	garr_betriebsmeldungen[st_config_achse.i16_meld_startindex + 0] := FALSE;
	garr_betriebsmeldungen[st_config_achse.i16_meld_startindex + 1] := FALSE;
	garr_betriebsmeldungen[st_config_achse.i16_meld_startindex + 2] := FALSE;
	garr_betriebsmeldungen[st_config_achse.i16_meld_startindex + 3] := FALSE;
	garr_betriebsmeldungen[st_config_achse.i16_meld_startindex + 4] := FALSE;
	garr_betriebsmeldungen[st_config_achse.i16_meld_startindex + 5] := FALSE;
	garr_betriebsmeldungen[st_config_achse.i16_meld_startindex + 6] := FALSE;
	garr_betriebsmeldungen[st_config_achse.i16_meld_startindex + 7] := FALSE;
	garr_betriebsmeldungen[st_config_achse.i16_meld_startindex + 8] := FALSE;
	garr_betriebsmeldungen[st_config_achse.i16_meld_startindex + 9] := FALSE;
	garr_betriebsmeldungen[st_config_achse.i16_meld_startindex + 10] := FALSE;
	garr_betriebsmeldungen[st_config_achse.i16_meld_startindex + 11] := FALSE;
	garr_betriebsmeldungen[st_config_achse.i16_meld_startindex + 12] := FALSE;
	garr_betriebsmeldungen[st_config_achse.i16_meld_startindex + 13] := FALSE;
	garr_betriebsmeldungen[st_config_achse.i16_meld_startindex + 14] := FALSE;
	garr_betriebsmeldungen[st_config_achse.i16_meld_startindex + 15] := FALSE;
	garr_betriebsmeldungen[st_config_achse.i16_meld_startindex + 16] := FALSE;
	garr_betriebsmeldungen[st_config_achse.i16_meld_startindex + 17] := FALSE;
	garr_betriebsmeldungen[st_config_achse.i16_meld_startindex + 18] := FALSE;
	garr_betriebsmeldungen[st_config_achse.i16_meld_startindex + 19] := FALSE;
	garr_betriebsmeldungen[st_config_achse.i16_meld_startindex + 20] := FALSE;
	garr_betriebsmeldungen[st_config_achse.i16_meld_startindex + 21] := FALSE;
	garr_betriebsmeldungen[st_config_achse.i16_meld_startindex + 22] := FALSE;
	garr_betriebsmeldungen[st_config_achse.i16_meld_startindex + 23] := FALSE;
	garr_betriebsmeldungen[st_config_achse.i16_meld_startindex + 24] := FALSE;
	garr_betriebsmeldungen[st_config_achse.i16_meld_startindex + 25] := FALSE;
	garr_betriebsmeldungen[st_config_achse.i16_meld_startindex + 26] := FALSE;
	garr_betriebsmeldungen[st_config_achse.i16_meld_startindex + 27] := FALSE;
	garr_betriebsmeldungen[st_config_achse.i16_meld_startindex + 28] := FALSE;
	garr_betriebsmeldungen[st_config_achse.i16_meld_startindex + 29] := FALSE;
	garr_betriebsmeldungen[st_config_achse.i16_meld_startindex + 30] := FALSE;
	garr_betriebsmeldungen[st_config_achse.i16_meld_startindex + 31] := FALSE;
	garr_betriebsmeldungen[st_config_achse.i16_meld_startindex + 32] := FALSE;
	garr_betriebsmeldungen[st_config_achse.i16_meld_startindex + 33] := FALSE;
	garr_betriebsmeldungen[st_config_achse.i16_meld_startindex + 34] := FALSE;
	garr_betriebsmeldungen[st_config_achse.i16_meld_startindex + 35] := FALSE;
	garr_betriebsmeldungen[st_config_achse.i16_meld_startindex + 36] := FALSE;
	garr_betriebsmeldungen[st_config_achse.i16_meld_startindex + 37] := FALSE;
	garr_betriebsmeldungen[st_config_achse.i16_meld_startindex + 38] := FALSE;
	garr_betriebsmeldungen[st_config_achse.i16_meld_startindex + 39] := FALSE;
	garr_betriebsmeldungen[st_config_achse.i16_meld_startindex + 40] := FALSE;
	garr_betriebsmeldungen[st_config_achse.i16_meld_startindex + 41] := FALSE;
	garr_betriebsmeldungen[st_config_achse.i16_meld_startindex + 42] := FALSE;
	garr_betriebsmeldungen[st_config_achse.i16_meld_startindex + 43] := FALSE;
	garr_betriebsmeldungen[st_config_achse.i16_meld_startindex + 44] := FALSE;
	garr_betriebsmeldungen[st_config_achse.i16_meld_startindex + 45] := FALSE;
	garr_betriebsmeldungen[st_config_achse.i16_meld_startindex + 46] := FALSE;
	garr_betriebsmeldungen[st_config_achse.i16_meld_startindex + 47] := FALSE;
	garr_betriebsmeldungen[st_config_achse.i16_meld_startindex + 48] := FALSE;
	garr_betriebsmeldungen[st_config_achse.i16_meld_startindex + 49] := FALSE;
END_IF
END_PROGRAM

(* POU Maschine1720/WT Transport/ST_WT_Transport_Warteposition_1720, ST *)
PROGRAM ST_WT_Transport_Warteposition_1720
VAR_INPUT
	st_config								: struct_config;
	st_ctrl_in								: struct_ctrl_in;
	e_station_vorher_in_anforderung			: BOOL := FALSE;
	e_station_vorher_in_abgegeben			: BOOL := FALSE;
END_VAR
VAR_IN_OUT
	st_visu								: struct_visu;
END_VAR
VAR_OUTPUT
	st_ctrl_out							: struct_ctrl_out;
	a_station_vorher_out_erlaubnis			: BOOL := FALSE;
	a_station_vorher_out_angekommen		: BOOL := FALSE;
END_VAR
VAR
	fb_ton_uez							: TON;
	fb_ton_wz							: TON;
	fb_ton_quitt							: TON;
	fb_ton_wt_auf_wartepos				: TON;
	fb_tof_wt_auf_wartepos					: TOF;
	fb_r_trig_start							: R_TRIG;
	fb_r_trig_wartepos						: R_TRIG;
	fb_r_trig_wartepos_verlassen			: R_TRIG;
	fb_state_entry							: ST_StateEntry;
	sm_wt_hat_wartepos_nicht_verlassen	: BOOL := FALSE;
	sm_wt_hat_wartepos_ueberfahren		: BOOL := FALSE;
	bm_warte_anforderung					: BOOL := FALSE;
	bm_warte_wt_an_stopper				: BOOL := FALSE;
	bm_warte_beladepos_frei				: BOOL := FALSE;

	e_wt_auf_wartepos					AT %I* : BOOL;
	e_wt_wartepos_verlassen				AT %I* : BOOL;
END_VAR
(* Zeiten *)
fb_ton_uez(IN:= , PT:= , Q=>  , ET=> );
fb_ton_wz(IN:= , PT:= , Q=> , ET=> );
fb_ton_quitt(IN:= , PT:= t#100ms, Q=> , ET=> );

fb_ton_wt_auf_wartepos(IN:= e_wt_auf_wartepos, PT:= t#200ms, Q=> , ET=> );
fb_tof_wt_auf_wartepos(IN:= e_wt_auf_wartepos, PT:= t#200ms, Q=> , ET=> );

(* Flanken *)
fb_r_trig_wartepos(CLK:= e_wt_auf_wartepos, Q=> );
fb_r_trig_wartepos_verlassen(CLK:= e_wt_wartepos_verlassen, Q=> );
fb_r_trig_start(CLK:= st_ctrl_in.b_start, Q=> );

(* ==================================Toplevel=================================== *)
IF fb_state_entry.i16_next_step > INIT AND fb_state_entry.i16_next_step < FEHLER THEN
	(* Allgemeine Fehler *)
	IF st_ctrl_in.b_stop THEN
		fb_state_entry.i16_next_step := STOP;
	ELSIF zyl_wt_stopper_einlauf.st_ctrl.out.b_fehler THEN
		fb_state_entry.i16_next_step := FEHLER;
	(* Zylinder im Handbetrieb *)
	ELSIF gi16_betriebsart = HAND AND
		st_visu.st_zyl.i16_nr_zyl_im_handbetrieb = zyl_wt_stopper_einlauf.fb.st_config.i16_identnummer
		THEN
			fb_state_entry.i16_next_step := FEHLER;
	END_IF
END_IF

(* ============================Haupt-Schrittkette================================ *)
fb_state_entry(
	i16_next_step:= , 
	i16_pos:= 1,
	s_debugtext:= ,
	E=> ,
	X=> , 
	i16_step=> ,
	i16_last_step=> );

CASE fb_state_entry.i16_step OF
(*=======================================================*)
	INIT_OBJ:
		IF st_config.b_config_fertig THEN
			fb_state_entry.i16_next_step := INIT;
		END_IF

(*=======================================================*)
	INIT:
		IF fb_state_entry.E THEN
			fb_ton_wz.IN := FALSE;
			fb_ton_uez.IN := FALSE;
			fb_ton_quitt.IN := FALSE;
			st_ctrl_out.b_fehler := FALSE;
			st_ctrl_out.b_bereit := FALSE;
			st_ctrl_out.b_fertig := FALSE;
			st_ctrl_out.b_kontroller_start := FALSE;
			zyl_wt_stopper_einlauf.st_ctrl.in.b_einfahren := FALSE;
			zyl_wt_stopper_einlauf.st_ctrl.in.b_ausfahren := FALSE;
			sm_wt_hat_wartepos_nicht_verlassen := FALSE;
			sm_wt_hat_wartepos_ueberfahren := FALSE;
			bm_warte_anforderung := FALSE;
			bm_warte_wt_an_stopper := FALSE;
			bm_warte_beladepos_frei := FALSE;
			a_station_vorher_out_erlaubnis := FALSE;
			a_station_vorher_out_angekommen := FALSE;
		END_IF

		(*-----------------------Weiterschaltbedingungen----------------------------*)
		IF st_ctrl_in.b_init THEN
			zyl_wt_stopper_einlauf.st_ctrl.in.b_quittieren := FALSE;
			fb_state_entry.i16_next_step := 20;
		END_IF

(*=======================================================*)
	20: (* Initialisierung: Einlaufstopper ausfahren *)
		IF fb_state_entry.E THEN
			zyl_wt_stopper_einlauf.st_ctrl.in.b_ausfahren := TRUE;
		END_IF

		(*-----------------------Weiterschaltbedingungen----------------------------*)
		IF zyl_wt_stopper_einlauf.st_ctrl.out.b_ausgefahren THEN
			zyl_wt_stopper_einlauf.st_ctrl.in.b_ausfahren := FALSE;
			fb_state_entry.i16_next_step :=  BEREIT;
		END_IF

(*=======================================================*)
	BEREIT:	(* Warte auf Start von Kontroller *)
		IF fb_state_entry.E THEN
			st_ctrl_out.b_bereit := TRUE;
			st_ctrl_out.b_fertig := TRUE;
		END_IF

	(*-----------------------Weiterschaltbedingungen----------------------------*)
		IF st_config.b_station_aktiv OR st_config.b_station_in_simulation THEN
			(* WT Transport aktiv oder in Simulation *)
			IF st_ctrl_in.b_start THEN
			(* WT Transport gestartet *)
				st_ctrl_out.b_fertig := FALSE;
				fb_state_entry.i16_next_step := 110;
			END_IF
		ELSE
			fb_state_entry.i16_next_step := 500;
		END_IF

(*=======================================================*)
	110: (* Statische WT-Abfrage auf Warteposition nach der Initialisierung *)
		IF fb_state_entry.E THEN
			st_ctrl_out.b_kontroller_start := TRUE;
		END_IF

		IF NOT e_station_vorher_in_abgegeben THEN
			a_station_vorher_out_angekommen := FALSE;
		END_IF

		(*-----------------------Weiterschaltbedingungen----------------------------*)
		IF e_wt_auf_wartepos THEN
			st_ctrl_out.b_kontroller_start := FALSE;
			fb_state_entry.i16_next_step := 140;
		ELSE	(* Kein WT da, deshalb einen holen *)
			st_ctrl_out.b_kontroller_start := FALSE;
			fb_state_entry.i16_next_step := 120;
		END_IF

(*=======================================================*)
	120: (* Kein WT da -> warte auf Anforderung von vorheriger Station *)
		IF fb_state_entry.E THEN
			st_ctrl_out.b_kontroller_start := TRUE;
			bm_warte_anforderung := TRUE;
		END_IF

		IF NOT e_station_vorher_in_abgegeben THEN
			a_station_vorher_out_angekommen := FALSE;
		END_IF

		(*-----------------------Weiterschaltbedingungen----------------------------*)
		IF e_station_vorher_in_anforderung THEN
			a_station_vorher_out_angekommen := FALSE;
			a_station_vorher_out_erlaubnis := TRUE;
			st_ctrl_out.b_kontroller_start := FALSE;
			bm_warte_anforderung := FALSE;
			fb_state_entry.i16_next_step := 130;
		END_IF

(*=======================================================*)
	130: (* Warte bis WT an Stopper angekommen ist *)
		IF fb_state_entry.E THEN
			st_ctrl_out.b_kontroller_start := TRUE;
			bm_warte_wt_an_stopper := TRUE;
		END_IF

		(*-----------------------Weiterschaltbedingungen----------------------------*)
		IF fb_r_trig_wartepos.Q THEN
			a_station_vorher_out_erlaubnis := FALSE;
			a_station_vorher_out_angekommen := TRUE;
			st_ctrl_out.b_kontroller_start := FALSE;
			fb_ton_uez.IN := FALSE;
			bm_warte_wt_an_stopper := FALSE;
			fb_state_entry.i16_next_step := 140;
		END_IF

(*=======================================================*)
	140: (* WT ist da - Warten bis Beladeposition auf Bestücktisch frei ist *)
		IF fb_state_entry.E THEN
			zyl_wt_stopper_einlauf.st_ctrl.in.b_ausfahren := FALSE;
			zyl_wt_stopper_einlauf.st_ctrl.in.b_einfahren := FALSE;
			bm_warte_beladepos_frei := TRUE;
		END_IF

		(*-----------------------Weiterschaltbedingungen----------------------------*)
		IF NOT ST_WT_Transport_Beladen_1720.e_wt_auf_beladepos AND NOT axis_z_achse.st_ctrl.in.b_start THEN
			bm_warte_beladepos_frei := FALSE;
			fb_state_entry.i16_next_step := 150;
		ELSIF e_wt_wartepos_verlassen THEN
			(* Warteposition wurde unerlaubterweise überfahren *)
			sm_wt_hat_wartepos_ueberfahren := TRUE;
			fb_state_entry.i16_next_step := FEHLER;
		END_IF

(*=======================================================*)
	150: (* Bestücktisch ist frei -> Einlaufstopper einfahren *)
		IF fb_state_entry.E THEN
			zyl_wt_stopper_einlauf.st_ctrl.in.b_einfahren := TRUE;
		END_IF

		(*-----------------------Weiterschaltbedingungen----------------------------*)
		IF zyl_wt_stopper_einlauf.st_ctrl.out.b_eingefahren THEN
			zyl_wt_stopper_einlauf.st_ctrl.in.b_einfahren := FALSE;
			fb_state_entry.i16_next_step := 160;
		END_IF

(*=======================================================*)
	160: (* WT fährt weiter - Überwachung starten *)
		IF fb_state_entry.E THEN
			fb_ton_uez.PT := t#5s;
 			fb_ton_uez.IN := TRUE;
			st_ctrl_out.b_kontroller_start := TRUE;
		END_IF

		(*-----------------------Weiterschaltbedingungen----------------------------*)
		IF fb_r_trig_wartepos_verlassen.Q THEN
			fb_ton_uez.IN := FALSE;
			st_ctrl_out.b_kontroller_start := FALSE;
			fb_state_entry.i16_next_step := 170;
		ELSIF fb_ton_uez.Q THEN
			sm_wt_hat_wartepos_nicht_verlassen := TRUE;
			fb_state_entry.i16_next_step := FEHLER;
		END_IF

(*=======================================================*)
	170: (* Einlaufstopper ausfahren *)
		IF fb_state_entry.E THEN
			fb_ton_wz.IN := TRUE;
			fb_ton_wz.PT := t#1s;
			zyl_wt_stopper_einlauf.st_ctrl.in.b_ausfahren := TRUE;
		END_IF

		(*-----------------------Weiterschaltbedingungen----------------------------*)
		IF zyl_wt_stopper_einlauf.st_ctrl.out.b_ausgefahren AND fb_ton_wz.Q THEN
			zyl_wt_stopper_einlauf.st_ctrl.in.b_ausfahren := FALSE;
			fb_state_entry.i16_next_step := BEREIT;
			fb_ton_wz.IN := FALSE;
		END_IF

(*=======================================================*)
	500: (* Einlaufstopper einfahren, damit WTs auf Bestücktisch geschoben werden können. *)
		IF fb_state_entry.E THEN
			zyl_wt_stopper_einlauf.st_ctrl.in.b_einfahren := TRUE;
		END_IF

		(*-----------------------Weiterschaltbedingungen----------------------------*)
		IF zyl_wt_stopper_einlauf.st_ctrl.out.b_eingefahren THEN
			zyl_wt_stopper_einlauf.st_ctrl.in.b_einfahren := FALSE;
			fb_state_entry.i16_next_step :=  510;
		END_IF

(*=======================================================*)
	510:	(* Warte auf Konfigurationsänderung *)

	(*-----------------------Weiterschaltbedingungen----------------------------*)
		IF st_config.b_station_aktiv OR st_config.b_station_in_simulation THEN
			(* WT Transport aktiv oder in Simulation *)
			fb_state_entry.i16_next_step := BEREIT;
		END_IF

(*=======================================================*)
	FEHLER:
		IF fb_state_entry.E THEN
			st_ctrl_out.b_fehler := TRUE;
			fb_ton_quitt.IN := FALSE;
			zyl_wt_stopper_einlauf.st_ctrl.in.b_quittieren := FALSE;

			a_station_vorher_out_erlaubnis := FALSE;
			a_station_vorher_out_angekommen := FALSE;
		END_IF

		(*-----------------------Weiterschaltbedingungen----------------------------*)
		IF st_ctrl_in.b_quitt AND NOT fb_state_entry.E THEN
			st_ctrl_out.b_fehler := FALSE;
			zyl_wt_stopper_einlauf.st_ctrl.in.b_quittieren := TRUE;
			fb_ton_quitt.IN := TRUE;
		END_IF

		IF fb_ton_quitt.Q THEN
			fb_ton_quitt.IN := FALSE;
			fb_state_entry.i16_next_step := INIT;
		END_IF

(*=======================================================*)
	STOP:
		IF fb_state_entry.E THEN
			fb_ton_quitt.IN := FALSE;
			st_ctrl_out.b_kontroller_start := FALSE;
			zyl_wt_stopper_einlauf.st_ctrl.in.b_quittieren := FALSE;
			a_station_vorher_out_erlaubnis := FALSE;
			a_station_vorher_out_angekommen := FALSE;
		END_IF

		(*-----------------------Weiterschaltbedingungen----------------------------*)
		IF st_ctrl_in.b_quitt AND NOT fb_state_entry.E THEN
			fb_ton_quitt.IN := TRUE;
			zyl_wt_stopper_einlauf.st_ctrl.in.b_quittieren := TRUE;
		END_IF

		IF fb_ton_quitt.Q THEN
			fb_ton_quitt.IN := FALSE;
			fb_state_entry.i16_next_step := INIT;
		END_IF
END_CASE

fb_state_entry(
	i16_next_step:= ,
	i16_pos:= 2,
	s_debugtext:= ,
	E=> ,
	X=> ,
	i16_step=> ,
	i16_last_step=> );

IF st_config.b_config_fertig THEN
	(* Fehlermeldungen ab dem Startindex in das globale Störmeldungsarray schreiben *)
	garr_stoermeldungen[st_config.i16_meld_startindex + 0] := sm_wt_hat_wartepos_nicht_verlassen;
	garr_stoermeldungen[st_config.i16_meld_startindex + 1] := sm_wt_hat_wartepos_ueberfahren;
	garr_stoermeldungen[st_config.i16_meld_startindex + 2] := FALSE;
	garr_stoermeldungen[st_config.i16_meld_startindex + 3] := FALSE;
	garr_stoermeldungen[st_config.i16_meld_startindex + 4] := FALSE;
	garr_stoermeldungen[st_config.i16_meld_startindex + 5] := FALSE;
	garr_stoermeldungen[st_config.i16_meld_startindex + 6] := FALSE;
	garr_stoermeldungen[st_config.i16_meld_startindex + 7] := FALSE;
	garr_stoermeldungen[st_config.i16_meld_startindex + 8] := FALSE;
	garr_stoermeldungen[st_config.i16_meld_startindex + 9] := FALSE;
	garr_stoermeldungen[st_config.i16_meld_startindex + 10] := FALSE;
	garr_stoermeldungen[st_config.i16_meld_startindex + 11] := FALSE;
	garr_stoermeldungen[st_config.i16_meld_startindex + 12] := FALSE;
	garr_stoermeldungen[st_config.i16_meld_startindex + 13] := FALSE;
	garr_stoermeldungen[st_config.i16_meld_startindex + 14] := FALSE;
	garr_stoermeldungen[st_config.i16_meld_startindex + 15] := FALSE;
	garr_stoermeldungen[st_config.i16_meld_startindex + 16] := FALSE;
	garr_stoermeldungen[st_config.i16_meld_startindex + 17] := FALSE;
	garr_stoermeldungen[st_config.i16_meld_startindex + 18] := FALSE;
	garr_stoermeldungen[st_config.i16_meld_startindex + 19] := FALSE;
	
	garr_betriebsmeldungen[st_config.i16_meld_startindex + 0] := bm_warte_anforderung;
	garr_betriebsmeldungen[st_config.i16_meld_startindex + 1] := bm_warte_wt_an_stopper;
	garr_betriebsmeldungen[st_config.i16_meld_startindex + 2] := bm_warte_beladepos_frei;
	garr_betriebsmeldungen[st_config.i16_meld_startindex + 3] := FALSE;
	garr_betriebsmeldungen[st_config.i16_meld_startindex + 4] := FALSE;
	garr_betriebsmeldungen[st_config.i16_meld_startindex + 5] := FALSE;
	garr_betriebsmeldungen[st_config.i16_meld_startindex + 6] := FALSE;
	garr_betriebsmeldungen[st_config.i16_meld_startindex + 7] := FALSE;
	garr_betriebsmeldungen[st_config.i16_meld_startindex + 8] := FALSE;
	garr_betriebsmeldungen[st_config.i16_meld_startindex + 9] := FALSE;
	garr_betriebsmeldungen[st_config.i16_meld_startindex + 10] := FALSE;
	garr_betriebsmeldungen[st_config.i16_meld_startindex + 11] := FALSE;
	garr_betriebsmeldungen[st_config.i16_meld_startindex + 12] := FALSE;
	garr_betriebsmeldungen[st_config.i16_meld_startindex + 13] := FALSE;
	garr_betriebsmeldungen[st_config.i16_meld_startindex + 14] := FALSE;
	garr_betriebsmeldungen[st_config.i16_meld_startindex + 15] := FALSE;
	garr_betriebsmeldungen[st_config.i16_meld_startindex + 16] := FALSE;
	garr_betriebsmeldungen[st_config.i16_meld_startindex + 17] := FALSE;
	garr_betriebsmeldungen[st_config.i16_meld_startindex + 18] := FALSE;
	garr_betriebsmeldungen[st_config.i16_meld_startindex + 19] := FALSE;
END_IF
END_PROGRAM

(* POU Gemeinsamkeiten17xx/Werkzeug/ST_WkzAbsicherung, ST *)
PROGRAM ST_WkzAbsicherung
VAR_INPUT
	st_config								: struct_config;
	st_ctrl_in								: struct_ctrl_in;
END_VAR
VAR_IN_OUT
	st_visu								: struct_visu;
END_VAR
VAR_OUTPUT
	st_ctrl_out							: struct_ctrl_out;
END_VAR
VAR
	fb_ton_wz							: TON;
	fb_ton_uez							: TON;
	fb_ton_quitt							: TON;
	fb_state_entry							: ST_StateEntry;
	b_signalmerker_bestueckschieber_on		: BOOL := FALSE;
	b_signalmerker_bestueckschieber_off		: BOOL := FALSE;
	fb_r_trig_signal_bestueckschieber		: R_TRIG;
	fb_f_trig_signal_bestueckschieber		: F_TRIG;
	fb_r_trig_nocke_uw_bestueckschieber	: R_TRIG;
	fb_f_trig_nocke_uw_bestueckschieber	: F_TRIG;

	(* Eingänge *)
	(* BSV 1720 6-fach *)
	e_wkz_sicherung_niederhalter_li			AT %I* : BOOL;
	e_wkz_sicherung_faenger_li			AT %I* : BOOL;
	e_wkz_sicherung_abfallpodest_li		AT %I* : BOOL;
	e_wkz_sicherung_niederhalter_re		AT %I* : BOOL;
	e_wkz_sicherung_faenger_re			AT %I* : BOOL;
	e_wkz_sicherung_abfallpodest_re		AT %I* : BOOL;
	(* Erkennung/Kodierung für alte WKZ z.B. 1708alt *)
	e_kodierung_alt_wkz					AT %I* : BOOL;
	(* BSH 1700 *)
	e_wkz_sicherung_faenger				AT %I* : BOOL;
	e_bestueckschieber_ueberwachung		AT %I* : BOOL;

	(* Meldungen *)
	(* BSV 1720 6-fach *)
	sm_wkz_sicherung_niederhalter_li		: BOOL := FALSE;
	sm_wkz_sicherung_faenger_li			: BOOL := FALSE;
	sm_wkz_sicherung_abfallpodest_li		: BOOL := FALSE;
	sm_wkz_sicherung_niederhalter_re		: BOOL := FALSE;
	sm_wkz_sicherung_faenger_re			: BOOL := FALSE;
	sm_wkz_sicherung_abfallpodest_re		: BOOL := FALSE;
	(* BSH 1700 *)
	sm_wkz_sicherung_faenger				: BOOL := FALSE;
	sm_bestueckschieber_ueberwachung	: BOOL := FALSE;
	UW_Bestueckschieber_on: BOOL;
END_VAR
(* Zeiten *)
fb_ton_wz(IN:= , PT:= , Q=>  , ET=> );
fb_ton_uez(IN:= , PT:= , Q=>  , ET=> );
fb_ton_quitt(IN:= , PT:= t#100ms, Q=> , ET=> );

(* Flanken *)

fb_f_trig_nocke_uw_bestueckschieber(CLK:= nockenschaltwerk_bestueckachse.fb.arr_spur[SP_UW_BESTUECKSCHIEBER_ON], Q=> );
fb_r_trig_nocke_uw_bestueckschieber(CLK:= nockenschaltwerk_bestueckachse.fb.arr_spur[SP_UW_BESTUECKSCHIEBER_ON], Q=> );
fb_r_trig_signal_bestueckschieber(CLK:= e_bestueckschieber_ueberwachung, Q=> );
fb_f_trig_signal_bestueckschieber(CLK:= e_bestueckschieber_ueberwachung, Q=> );

UW_Bestueckschieber_on:=nockenschaltwerk_bestueckachse.fb.arr_spur[SP_UW_BESTUECKSCHIEBER_ON]; 	(*für Trace*)
(* Toplevel *)
IF fb_state_entry.i16_next_step > INIT AND fb_state_entry.i16_next_step < FEHLER THEN
	IF fb_state_entry.i16_next_step < STOP THEN
		IF st_ctrl_in.b_stop THEN
			fb_state_entry.i16_next_step := STOP;
		END_IF
	END_IF
END_IF

(* ======================================Schrittkette======================================== *)
fb_state_entry(
	i16_next_step:= ,
	i16_pos:= 1,
	s_debugtext:= ,
	E=> ,
	X=> ,
	i16_step=> ,
	i16_last_step=> );

CASE fb_state_entry.i16_step OF
(*=======================================================*)
	INIT_OBJ:
		IF st_config.b_config_fertig THEN
			fb_state_entry.i16_next_step := INIT;
		END_IF

(*=======================================================*)
	INIT:
		IF fb_state_entry.E THEN
			fb_ton_wz.IN := FALSE;
			fb_ton_uez.IN	:= FALSE;
			fb_ton_quitt.IN	 := FALSE;
			b_signalmerker_bestueckschieber_on := FALSE;
			b_signalmerker_bestueckschieber_off := FALSE;
			sm_wkz_sicherung_niederhalter_li := FALSE;
			sm_wkz_sicherung_faenger_li := FALSE;
			sm_wkz_sicherung_abfallpodest_li := FALSE;
			sm_wkz_sicherung_niederhalter_re := FALSE;
			sm_wkz_sicherung_faenger_re := FALSE;
			sm_wkz_sicherung_abfallpodest_re := FALSE;
			sm_wkz_sicherung_faenger := FALSE;
			sm_bestueckschieber_ueberwachung := FALSE;
			st_ctrl_out.b_fehler := FALSE;
			st_ctrl_out.b_bereit := FALSE;
			st_ctrl_out.b_fertig := FALSE;
			st_ctrl_out.b_einzelfertigung := FALSE;
		END_IF

		(*-----------------------Weiterschaltbedingungen----------------------------*)
		IF st_ctrl_in.b_init THEN
			fb_state_entry.i16_next_step := BEREIT;
		END_IF

(*=======================================================*)
	BEREIT:
		IF fb_state_entry.E THEN
			st_ctrl_out.b_bereit := TRUE;
		END_IF

		CASE gst_datensatz.st_md.i16_typ_zelle OF
			KEINE_ZELLE:
				;

			BESTUECKZELLE_1700:
				IF NOT gst_datensatz.st_md.b_wt_transport_simulation THEN
					IF NOT e_wkz_sicherung_faenger THEN
						sm_wkz_sicherung_faenger := TRUE;
						fb_state_entry.i16_next_step := FEHLER;
					END_IF

					IF ST_Virtuelle_Masterachse.fb_state_entry.i16_step >= BEREIT THEN
						IF gst_datensatz.st_bestueckprogramm.i16_b[ST_Virtuelle_Masterachse.i16_bestueckposzaehler] <> 0 THEN	(* Bei Umfahrung = 0 bewegt sich der Bestückschieber nicht *)
							(* Nocken werden in virtueller Bestückachse nach ein paar Hüben ausgeschaltet *)
							IF	(nockenschaltwerk_bestueckachse.fb.arr_spur[SP_UW_BESTUECKSCHIEBER_ON] AND  NOT e_bestueckschieber_ueberwachung) OR
								(nockenschaltwerk_bestueckachse.fb.arr_spur[SP_UW_BESTUECKSCHIEBER_OFF] AND e_bestueckschieber_ueberwachung)
								THEN
									sm_bestueckschieber_ueberwachung := TRUE;
									fb_state_entry.i16_next_step := FEHLER;
							END_IF
						END_IF
					END_IF


					(* Option: Flankenauswertung der GLS am Bestückschieber *)
(*					IF	nockenschaltwerk_bestueckachse.fb.arr_spur[SP_UW_BESTUECKSCHIEBER_ON] THEN
						IF 	fb_r_trig_signal_bestueckschieber.Q THEN
							b_signalmerker_bestueckschieber_on := TRUE;
						END_IF
						IF	 fb_f_trig_signal_bestueckschieber.Q THEN
							b_signalmerker_bestueckschieber_off := TRUE;
						END_IF
					END_IF

					(* Option: Beide setzen wenn Nocke abgeschaltet ist *)
					IF	NOT gst_datensatz.st_wkz.nockenschaltwerk_bestueckachse.arr_nocken[SP_UW_BESTUECKSCHIEBER_OFF].b_camvalid THEN
						b_signalmerker_bestueckschieber_on := TRUE;
						b_signalmerker_bestueckschieber_off := TRUE;
					END_IF

					IF 	fb_f_trig_nocke_uw_bestueckschieber.Q THEN

						IF 	b_signalmerker_bestueckschieber_off  AND
							b_signalmerker_bestueckschieber_on THEN
							b_signalmerker_bestueckschieber_on := FALSE;
							b_signalmerker_bestueckschieber_off := FALSE;
						ELSE
							sm_bestueckschieber_ueberwachung := TRUE;
							fb_state_entry.i16_next_step := FEHLER;
						END_IF
					END_IF
*)
				END_IF

			BESTUECKZELLE_1720:
				IF NOT gst_datensatz.st_md.b_wt_transport_simulation THEN
					IF e_kodierung_alt_wkz THEN
						(* BSV 1720 2-fach *)
						IF NOT  e_wkz_sicherung_faenger_li THEN
							sm_wkz_sicherung_faenger_li := TRUE;
							fb_state_entry.i16_next_step := FEHLER;
						END_IF
						IF NOT  e_wkz_sicherung_faenger_re THEN
							sm_wkz_sicherung_faenger_re := TRUE;
							fb_state_entry.i16_next_step := FEHLER;
						END_IF
					ELSE
						(* BSV 1720 6-fach *)
						IF	NOT ST_TippTasten.b_einfaedeln_aktiv THEN
							IF e_wkz_sicherung_niederhalter_li AND nockenschaltwerk_bestueckachse.fb.arr_spur[SP_UW_WKZ_NIEDERHALTER_LI] THEN
								sm_wkz_sicherung_niederhalter_li := TRUE;
								fb_state_entry.i16_next_step := 200;
							END_IF
							IF e_wkz_sicherung_niederhalter_re AND nockenschaltwerk_bestueckachse.fb.arr_spur[SP_UW_WKZ_NIEDERHALTER_RE] THEN
								sm_wkz_sicherung_niederhalter_re := TRUE;
								fb_state_entry.i16_next_step := 200;
							END_IF
						END_IF
						IF NOT  e_wkz_sicherung_faenger_li THEN
							sm_wkz_sicherung_faenger_li := TRUE;
							fb_state_entry.i16_next_step := FEHLER;
						END_IF
						IF NOT  e_wkz_sicherung_faenger_re THEN
							sm_wkz_sicherung_faenger_re := TRUE;
							fb_state_entry.i16_next_step := FEHLER;
						END_IF
						IF NOT e_wkz_sicherung_abfallpodest_li THEN
							sm_wkz_sicherung_abfallpodest_li := TRUE;
							fb_state_entry.i16_next_step := 200;
						END_IF
						IF NOT e_wkz_sicherung_abfallpodest_re THEN
							sm_wkz_sicherung_abfallpodest_re := TRUE;
							fb_state_entry.i16_next_step := 200;
						END_IF
					END_IF
				END_IF

			RASTERFOLIE:
				;
		END_CASE

(*=======================================================*)
	200:	(* Nur aktiv bei 1720 und WKZ-Absicherung 6-fach. Verzweigen nach Fehler erst, wenn OT erreicht wird - leichtere Fehlerbehebung. *)

		IF NOT gst_datensatz.st_md.b_wt_transport_simulation THEN
			(* BSV 1720 6-fach *)
			IF e_wkz_sicherung_niederhalter_li AND nockenschaltwerk_bestueckachse.fb.arr_spur[SP_UW_WKZ_NIEDERHALTER_LI] THEN
				sm_wkz_sicherung_niederhalter_li := TRUE;
			END_IF
			IF NOT  e_wkz_sicherung_faenger_li THEN
				sm_wkz_sicherung_faenger_li := TRUE;
				fb_state_entry.i16_next_step := FEHLER;
			END_IF
			IF NOT e_wkz_sicherung_abfallpodest_li THEN
				sm_wkz_sicherung_abfallpodest_li := TRUE;
			END_IF
			IF e_wkz_sicherung_niederhalter_re AND nockenschaltwerk_bestueckachse.fb.arr_spur[SP_UW_WKZ_NIEDERHALTER_RE] THEN
				sm_wkz_sicherung_niederhalter_re := TRUE;
			END_IF
			IF NOT  e_wkz_sicherung_faenger_re THEN
				sm_wkz_sicherung_faenger_re := TRUE;
				fb_state_entry.i16_next_step := FEHLER;
			END_IF
			IF NOT e_wkz_sicherung_abfallpodest_re THEN
				sm_wkz_sicherung_abfallpodest_re := TRUE;
			END_IF
		END_IF

		(*-----------------------Weiterschaltbedingungen----------------------------*)
		IF nockenschaltwerk_bestueckachse.fb.arr_spur[SP_OT]  THEN
			fb_state_entry.i16_next_step := FEHLER;
		END_IF

(*=======================================================*)
	FEHLER:
		IF fb_state_entry.E THEN
			st_ctrl_out.b_fehler := TRUE;
			fb_ton_quitt.IN := FALSE;
		END_IF

		(*-----------------------Weiterschaltbedingungen----------------------------*)
		IF st_ctrl_in.b_quitt AND NOT fb_state_entry.E THEN
			st_ctrl_out.b_fehler := FALSE;
			fb_ton_quitt.IN := TRUE;
		END_IF

		IF fb_ton_quitt.Q THEN
			fb_ton_quitt.IN := FALSE;
			fb_state_entry.i16_next_step := INIT;
		END_IF

(*=======================================================*)
	STOP:
		IF fb_state_entry.E THEN
			fb_ton_quitt.IN := FALSE;
		END_IF

		(*-----------------------Weiterschaltbedingungen----------------------------*)
		IF st_ctrl_in.b_quitt AND NOT fb_state_entry.E THEN
			fb_ton_quitt.IN := TRUE;
		END_IF

		IF fb_ton_quitt.Q THEN
			fb_ton_quitt.IN := FALSE;
			fb_state_entry.i16_next_step := INIT;
		END_IF
END_CASE

fb_state_entry(
	i16_next_step:= , 
	i16_pos:= 2,
	s_debugtext:= ,
	E=> , 
	X=> , 
	i16_step=> ,
	i16_last_step=> );

IF st_config.b_config_fertig THEN
	(* Fehlermeldungen und Betriebsmeldungen ab dem Startindex in die globalen Meldungsarrays schreiben *)
	garr_stoermeldungen[st_config.i16_meld_startindex + 0] := sm_wkz_sicherung_faenger;
	garr_stoermeldungen[st_config.i16_meld_startindex + 1] := sm_bestueckschieber_ueberwachung;
	garr_stoermeldungen[st_config.i16_meld_startindex + 2] := FALSE;
	garr_stoermeldungen[st_config.i16_meld_startindex + 3] := FALSE;
	garr_stoermeldungen[st_config.i16_meld_startindex + 4] := sm_wkz_sicherung_niederhalter_li;
	garr_stoermeldungen[st_config.i16_meld_startindex + 5] := sm_wkz_sicherung_faenger_li;
	garr_stoermeldungen[st_config.i16_meld_startindex + 6] := sm_wkz_sicherung_abfallpodest_li;
	garr_stoermeldungen[st_config.i16_meld_startindex + 7] := FALSE;
	garr_stoermeldungen[st_config.i16_meld_startindex + 8] := sm_wkz_sicherung_niederhalter_re;
	garr_stoermeldungen[st_config.i16_meld_startindex + 9] := sm_wkz_sicherung_faenger_re;
	garr_stoermeldungen[st_config.i16_meld_startindex + 10] := sm_wkz_sicherung_abfallpodest_re;
	garr_stoermeldungen[st_config.i16_meld_startindex + 11] := FALSE;
	garr_stoermeldungen[st_config.i16_meld_startindex + 12] := FALSE;
	garr_stoermeldungen[st_config.i16_meld_startindex + 13] := FALSE;
	garr_stoermeldungen[st_config.i16_meld_startindex + 14] := FALSE;
	garr_stoermeldungen[st_config.i16_meld_startindex + 15] := FALSE;
	garr_stoermeldungen[st_config.i16_meld_startindex + 16] := FALSE;
	garr_stoermeldungen[st_config.i16_meld_startindex + 17] := FALSE;
	garr_stoermeldungen[st_config.i16_meld_startindex + 18] := FALSE;
	garr_stoermeldungen[st_config.i16_meld_startindex + 19] := FALSE;
	
	garr_betriebsmeldungen[st_config.i16_meld_startindex + 0] := FALSE;
	garr_betriebsmeldungen[st_config.i16_meld_startindex + 1] := FALSE;
	garr_betriebsmeldungen[st_config.i16_meld_startindex + 2] := FALSE;
	garr_betriebsmeldungen[st_config.i16_meld_startindex + 3] := FALSE;
	garr_betriebsmeldungen[st_config.i16_meld_startindex + 4] := FALSE;
	garr_betriebsmeldungen[st_config.i16_meld_startindex + 5] := FALSE;
	garr_betriebsmeldungen[st_config.i16_meld_startindex + 6] := FALSE;
	garr_betriebsmeldungen[st_config.i16_meld_startindex + 7] := FALSE;
	garr_betriebsmeldungen[st_config.i16_meld_startindex + 8] := FALSE;
	garr_betriebsmeldungen[st_config.i16_meld_startindex + 9] := FALSE;
	garr_betriebsmeldungen[st_config.i16_meld_startindex + 10] := FALSE;
	garr_betriebsmeldungen[st_config.i16_meld_startindex + 11] := FALSE;
	garr_betriebsmeldungen[st_config.i16_meld_startindex + 12] := FALSE;
	garr_betriebsmeldungen[st_config.i16_meld_startindex + 13] := FALSE;
	garr_betriebsmeldungen[st_config.i16_meld_startindex + 14] := FALSE;
	garr_betriebsmeldungen[st_config.i16_meld_startindex + 15] := FALSE;
	garr_betriebsmeldungen[st_config.i16_meld_startindex + 16] := FALSE;
	garr_betriebsmeldungen[st_config.i16_meld_startindex + 17] := FALSE;
	garr_betriebsmeldungen[st_config.i16_meld_startindex + 18] := FALSE;
	garr_betriebsmeldungen[st_config.i16_meld_startindex + 19] := FALSE;
END_IF
END_PROGRAM

(* POU EPT Lib/Funktionen/DT_TO_SPECIALSTRING_YYYY_MM, ST *)
FUNCTION DT_TO_SPECIALSTRING_YYYY_MM : STRING
VAR_INPUT
	inDT					:	DT;
END_VAR
VAR

	TempString		:	STRING;
	SysTime				:	TIMESTRUCT;


	wYear					: WORD;
	wMonth				: WORD;
	wDay					: WORD;
	wHour					: WORD;
	wMin					: WORD;
	wSec					: WORD;
END_VAR
(*gVarStrSystemTime:=SYSTEMTIME_TO_STRING(gFB_GETLOCALSYSTEMTIME.systemTime);
gVarDTSystemtime:=SYSTEMTIME_TO_DT(gFB_GETLOCALSYSTEMTIME.SystemTime);
gVarSystemtime:=gFB_GETLOCALSYSTEMTIME.systemTime;
*)

SysTime:=DT_TO_SYSTEMTIME(inDT);

wYear:=SysTime.wYear;
wMonth:=SysTime.wMonth;
wDay:=SysTime.wDay;
wHour:=SysTime.wHour;
wMin:=SysTime.wMinute;
wSec:=SysTime.wSecond;
TempString:='';

TempString:=CONCAT(TempString ,WORD_TO_STRING(wYear));
TempString:=CONCAT(TempString ,'_');

IF wMonth<10 THEN	TempString:=CONCAT(TempString ,WORD_TO_STRING(0)); END_IF;
TempString:=CONCAT(TempString ,WORD_TO_STRING(wMonth));


DT_TO_SPECIALSTRING_YYYY_MM:=TempString;
END_FUNCTION

(* POU Gemeinsamkeiten17xx/Allgemeines/ST_Gesamthubzaehler, ST *)
PROGRAM ST_Gesamthubzaehler
VAR
	fb_tp_wz				: TP;
	fb_r_trig				: R_TRIG;
	a_Gesamthubzaehler	 AT %Q* : BOOL;
END_VAR
(* Erzeugung eines zeitkonstanten Zählersignals *)
fb_tp_wz(IN:= nockenschaltwerk_bestueckachse.fb.arr_spur[SP_OT], PT:= t#20ms, Q=> a_Gesamthubzaehler, ET=> );

(* Interner Bestückhubzähler der Maschine*)
fb_r_trig(CLK:= nockenschaltwerk_bestueckachse.fb.arr_spur[SP_OT], Q=> );

IF fb_r_trig.Q THEN
	gst_datensatz.st_md.i32_bestueckhubzaehler := gst_datensatz.st_md.i32_bestueckhubzaehler + 1;
	gst_datensatz.st_md.i32_werkzeughubzaehler := 	gst_datensatz.st_md.i32_werkzeughubzaehler +1;
END_IF

IF gst_datensatz.st_md.i32_bestueckhubzaehler > (EXPT(2,32)) OR gst_datensatz.st_md.i32_bestueckhubzaehler < 0 THEN
	gst_datensatz.st_md.i32_bestueckhubzaehler := 0;
END_IF
END_PROGRAM

(* POU Gemeinsamkeiten17xx/Allgemeines/ST_LampeMaterialMangel, ST *)
PROGRAM ST_LampeMaterialMangel
VAR_INPUT
	b_materialmangel		: ARRAY[0..7] OF BOOL;
END_VAR
VAR
	a_Lampe			AT %Q* : BOOL;
	fb_blinker			: ST_Blinker;
END_VAR
(* Blinken *)
(*schnell*)
IF 	b_materialmangel[1] 	THEN	(*Öl leer*)
fb_blinker(
	b_start:= TRUE,
	t_taktzeit_on:=t#500ms,
	t_taktzeit_off:=t#500ms,
	b_blinker_out=> );
END_IF
(*langsam*)
IF 	NOT b_materialmangel[1] AND	(*Öl leer*)
	( b_materialmangel[2] OR b_materialmangel[6] ) THEN	(*Stufe kleiner 10 or Korrektur X-Y zu hoch*)
fb_blinker(
	b_start:= TRUE,
	t_taktzeit_on:=t#1500ms,
	t_taktzeit_off:=t#1500ms,
	b_blinker_out=> );
END_IF


(* Materialmangel ist eingetreten *)
IF 	b_materialmangel[0] OR	(*Band leer*)
	b_materialmangel[1] OR	(*Öl leer*)
	b_materialmangel[2] OR	(*Stufe kleiner 10*)
	b_materialmangel[3] OR	(* Bandwechsel *)
	b_materialmangel[4] OR	(*Schaltschrank Temp*)
	b_materialmangel[5] OR	(* Band nicht abgescannt *)
	b_materialmangel[6] 		(* Korrektur X-Y Wert zu hoch *)
	THEN
		a_Lampe := fb_blinker.b_blinker_out OR b_materialmangel[0] OR b_materialmangel[3];

(* Es liegt kein Materialmangel vor *)
ELSE
	a_Lampe := FALSE;
END_IF
END_PROGRAM

(* POU EPT Lib/Funktionsbausteine/ST_Blinker, ST *)
FUNCTION_BLOCK ST_Blinker
VAR_INPUT
	b_start 		: BOOL;
	t_taktzeit_on	: TIME;
	t_taktzeit_off	: TIME;
END_VAR
VAR_OUTPUT
	b_blinker_out : BOOL;
END_VAR
VAR
	ton_on		: TON;
	ton_off		: TON;
END_VAR
ton_on(IN:=b_start AND NOT ton_off.Q , PT:=t_taktzeit_on , Q=>b_blinker_out , ET=> );
ton_off(IN:= ton_on.Q  , PT:=t_taktzeit_off , Q=> , ET=> );
END_FUNCTION_BLOCK

(* POU Gemeinsamkeiten17xx/Allgemeines/ST_Scope, ST *)
PROGRAM ST_Scope
VAR
	fb_ton_wz			: TON;
	fb_r_trig_bereit		: R_TRIG;
	fb_state_entry			: ST_StateEntry;

	fb_ScopeStop		: ScopeSetOffline;
	fb_ScopeOnline		: ScopeSetOnline;
	fb_ScopeExport		: ScopeViewExport;

	b_Stop				: BOOL;
	s_file_name			: STRING;
	pos					: INT;
	i					: INT;
	i32_error_id			:UDINT;
END_VAR

VAR CONSTANT
	s_path				: STRING:='C:\TwinCAT\Scope\';
END_VAR
(*===============================================================
   PRG: ST_Scope
  ---------------------------------------------------------------
   Auth: 		Werner Friedl
   Date: 		03.08.2016    						    
   Rev.: 		1.0
   Beschreibung:
	Mit diesem Programm wird das Scope automatisch gestartet und bei einem Fehler 
	ein Scopedatei mit aktueller Zeit im Verzeichnis "C:\TwinCAT\Scope\" abgespeichert. 

	-	zuerst muss ein Scope geöffnet und ein Projekt erstellt werden.
	-	Fehler für Stop eintragen	
	-	ST_ScopeStop startet das Scope bei "Anlage betriebsbereit"
	-	bei Fehler wird die Aufzeichnung nach 2sec gestoppt
	-	Auzeichnung	wird mit aktueller Zeit abgespeichert.	

hier Fehler für Stop einfügen============================================*)
(*b_Stop:=	ST_Bestueckachse.st_ctrl_out.b_fehler  OR
		axis_bestueckachse.st_ctrl.out.b_fehler ;*)

b_Stop:= (gi16_maschinenstatusinfo = STATUS_FEHLER);

(*=======================================================*)
fb_ton_wz(IN:=,PT:=T#2s);
fb_r_trig_bereit(CLK:= gi16_maschinenstatusinfo = STATUS_BETRIEBSBEREIT, Q=> );
fb_ScopeStop(bExecute:= , bBusy=> , bError=> , iErrorId=> );
fb_ScopeOnline(bExecute:= , bBusy=> , bError=> , iErrorId=> );
fb_ScopeExport(bExecute:=, sFilePath:=, tTimeout:=T#5s);

(*=======================================================*)
fb_state_entry(i16_pos:= 1, );

CASE fb_state_entry.i16_step OF
(*=======================================================*)
	INIT_OBJ:
		fb_state_entry.i16_next_step := INIT;

(*=======================================================*)
	INIT:
		IF	fb_state_entry.E THEN
			fb_ScopeOnline.bExecute:=FALSE;
			fb_ScopeStop.bExecute:=FALSE;
			fb_ScopeExport.bExecute:=FALSE;
		END_IF

		fb_state_entry.i16_next_step := BEREIT;


(*=======================================================*)
	BEREIT: (*warten auf betriebsbereit *)
		IF	fb_state_entry.E THEN
			b_Stop:=FALSE;
		END_IF

		IF	fb_r_trig_bereit.Q THEN
			fb_state_entry.i16_next_step := 110;
		END_IF


(*=======================================================*)
	110: (* Scope starten *)
		IF 	fb_state_entry.E THEN
			fb_ScopeOnline.bExecute:=TRUE;
		END_IF

		(*-----------------------Weiterschaltbedingungen----------------------------*)
		IF	fb_ScopeOnline.bBusy THEN
			fb_state_entry.i16_next_step := 120;
		END_IF

(*=======================================================*)
	120: (* Scope starten *)

		IF	NOT fb_ScopeOnline.bBusy THEN
			fb_state_entry.i16_next_step := 130;
			fb_ScopeOnline.bExecute:=FALSE;
		END_IF

		IF	fb_ScopeOnline.bError THEN
			i32_error_id:=fb_ScopeOnline.iErrorId;
			fb_state_entry.i16_next_step := FEHLER;
		END_IF

(*=======================================================*)
	130: (* warten auf Fehler *)
		IF	 fb_state_entry.E THEN
			fb_ton_wz.IN:=FALSE;
		END_IF

		fb_ton_wz.IN:=b_Stop ;
		fb_ScopeStop.bExecute:=fb_ton_wz.Q;


		IF	fb_ScopeStop.bBusy THEN
			fb_state_entry.i16_next_step := 140;
		END_IF

		IF	 fb_state_entry.X THEN
			fb_ton_wz.IN:=FALSE;
		END_IF
(*=======================================================*)
	140: (* Scope anhalten *)

		IF	NOT fb_ScopeStop.bBusy THEN
			fb_ScopeStop.bExecute:=FALSE;
			fb_state_entry.i16_next_step := 150;
		END_IF

		IF	fb_ScopeStop.bError THEN
			i32_error_id:=fb_ScopeStop.iErrorId;
			fb_state_entry.i16_next_step := FEHLER;
		END_IF

(*=======================================================*)
	150: (* Scope speichern *)
		IF 	fb_state_entry.E THEN
			s_file_name:=gstr_system_time;
			i:=0;
			FOR i := 1 TO 5  BY 1DO
				pos:=0;
				pos:=FIND(s_file_name,':');
				IF	pos > 0 THEN
					s_file_name:=REPLACE(s_file_name,'-',1,pos);
				END_IF
			END_FOR

			s_file_name:=CONCAT(s_file_name,'_Scope_View');
			s_file_name:=CONCAT(s_file_name,'.svw');

			fb_ScopeExport.sFilePath:=CONCAT(s_path,s_file_name);
			fb_ScopeExport.bExecute:=TRUE;
		END_IF

		(*-----------------------Weiterschaltbedingungen----------------------------*)
		IF	fb_ScopeExport.bBusy THEN
			fb_state_entry.i16_next_step := 160;
		END_IF


(*=======================================================*)
	160: (* Scope speichern *)

		IF	NOT fb_ScopeExport.bBusy THEN
			fb_state_entry.i16_next_step := BEREIT;
			fb_ScopeExport.bExecute:=FALSE;
		END_IF

		IF	fb_ScopeExport.bError THEN
			i32_error_id:=fb_ScopeExport.iErrorId;
			fb_state_entry.i16_next_step := FEHLER;
		END_IF

(*=======================================================*)
	FEHLER:	(*bei Fehler einfach weiter*)
		IF 	fb_state_entry.E THEN
			;
		END_IF
			fb_state_entry.i16_next_step := INIT;

END_CASE

fb_state_entry(i16_pos:= 2 );
END_PROGRAM

(* POU Gemeinsamkeiten17xx/Allgemeines/ST_Tuerverriegelung, ST *)
PROGRAM ST_Tuerverriegelung
VAR_INPUT
	e_quittiertaste						: BOOL;
END_VAR
VAR
	fb_ton_wz						: TON;
	fb_r_trig_quitt						: R_TRIG;
	fb_f_trig_quitt						: F_TRIG;
	fb_blinker						: ST_Blinker;
	a_tuerverriegelung_vorne			AT %Q* : BOOL;
	a_tuerverriegelung_hinten			AT %Q* : BOOL;
	e_kontakt_tuerverriegelung_vorne	AT %I* : BOOL;
	e_kontakt_tuerverriegelung_hinten	AT %I* : BOOL;
END_VAR
(* Blinken *)
fb_blinker(
	b_start:= TRUE,
	t_taktzeit_on:=t#500ms,
	t_taktzeit_off:=t#500ms,
	b_blinker_out=> );

(* Zeiten *)
fb_ton_wz(IN:= , PT:= t#3s, Q=> , ET=> );

(* Flanken *)
fb_r_trig_quitt(CLK:= e_quittiertaste, Q=> );
fb_f_trig_quitt(CLK:= e_quittiertaste, Q=> );

(* Ansteuerung der Türverriegelung vorne und hinten *)
CASE gi16_betriebsart OF
	HAND:
		a_tuerverriegelung_vorne := FALSE;
		a_tuerverriegelung_hinten := FALSE;
	TIPPEN, AUTO:
		IF 	gi16_maschinenstatusinfo = STATUS_BETRIEBSBEREIT OR
			gi16_maschinenstatusinfo = STATUS_FEHLER
			THEN
				(* Türen freigeben *)
				a_tuerverriegelung_vorne := FALSE;
				a_tuerverriegelung_hinten := FALSE;
		ELSE
			(* Türen verriegelt, wenn geschlossen *)
			IF NOT e_kontakt_tuerverriegelung_vorne THEN
				a_tuerverriegelung_vorne := TRUE;
			END_IF
			IF NOT e_kontakt_tuerverriegelung_hinten THEN
				a_tuerverriegelung_hinten := TRUE;
			END_IF
		END_IF
END_CASE
END_PROGRAM

(* POU Gemeinsamkeiten17xx/Bandeinzug/ST_Anwahl_Bandeinzug, ST *)
PROGRAM ST_Anwahl_Bandeinzug
VAR
	b_first_cycle 						: BOOL := TRUE;
	i16_typ_bandeinzug_visu			: enum_typ_bandeinzug_visu := KEIN_BANDEINZUG;
END_VAR
(*======================================================
   PRG: ExportResultString
 ------------------------------------------------------
   Auth: 		Werner Friedl    						 
   Date: 		07.03.2016    						     
   Rev.: 		1.0	
   Desc:		Damit bei unterschiedlichen Zellen (1700 oder 1720) nur die vorhandenen Bandwechsler in der Visu vorne angezeigt werden,
			müssen diese der Struktur "i16_typ_bandeinzug" zugewiesen werden.
   Historie:   1.0

 ========================================================*)
IF 	gi16_bbgen_auftrag = LESE_WKZ THEN
	b_first_cycle:=TRUE;
END_IF



IF	NOT b_first_cycle THEN

	CASE gst_datensatz.st_md.i16_typ_zelle OF
		KEINE_ZELLE:
			;

		BESTUECKZELLE_1700, RASTERFOLIE:
	
			CASE i16_typ_bandeinzug_visu OF

				KEIN_BANDEINZUG :
						gst_datensatz.st_wkz.i16_typ_bandeinzug:=KEIN_EINZUG;					;
				BANDEINZUG_1:
						gst_datensatz.st_wkz.i16_typ_bandeinzug:=BANDWECHSLER_V2;
				BANDEINZUG_2:
						gst_datensatz.st_wkz.i16_typ_bandeinzug:=SERVO;
				BANDEINZUG_3:
					;
			END_CASE

		BESTUECKZELLE_1720:

			CASE i16_typ_bandeinzug_visu OF
	
				KEIN_BANDEINZUG :
						gst_datensatz.st_wkz.i16_typ_bandeinzug:=KEIN_EINZUG;
				BANDEINZUG_1:
						gst_datensatz.st_wkz.i16_typ_bandeinzug:=STANDARD_2FACH_V2;
				BANDEINZUG_2:
					;
				BANDEINZUG_3:
					;
			END_CASE

	END_CASE

ELSIF	 gi16_bbgen_auftrag = KEIN_BB_AUFTRAG AND b_first_cycle THEN

	CASE gst_datensatz.st_md.i16_typ_zelle OF
		KEINE_ZELLE:
			;

		BESTUECKZELLE_1700, RASTERFOLIE:

			CASE gst_datensatz.st_wkz.i16_typ_bandeinzug OF

				KEIN_EINZUG :
					i16_typ_bandeinzug_visu:=KEIN_BANDEINZUG;
				BANDWECHSLER_V2:
					i16_typ_bandeinzug_visu:=BANDEINZUG_1;
				SERVO:
					i16_typ_bandeinzug_visu:=BANDEINZUG_2;

			END_CASE
			b_first_cycle:=FALSE;

		BESTUECKZELLE_1720:
	
			CASE gst_datensatz.st_wkz.i16_typ_bandeinzug OF

				KEIN_EINZUG :
					i16_typ_bandeinzug_visu:=KEIN_BANDEINZUG;
				STANDARD_2FACH_V2:
					i16_typ_bandeinzug_visu:=BANDEINZUG_1;

			END_CASE
			b_first_cycle:=FALSE;

	END_CASE


END_IF
END_PROGRAM

(* POU Gemeinsamkeiten17xx/Betriebsfreigaben/ST_Betriebsfreigaben, ST *)
PROGRAM ST_Betriebsfreigaben
VAR_INPUT
	st_config							: struct_config;
	st_ctrl_in							: struct_ctrl_in;
	b_lampe_stoerung				: BOOL;
	b_lampe_produktion				: BOOL;
	e_steuerung_ein					: BOOL;
END_VAR
VAR_OUTPUT
	st_ctrl_out						: struct_ctrl_out;
END_VAR
VAR
	fb_tof_druck						: TOF;
	fb_tof_druck_hublift_links			: TOF;
	fb_ton_ls_schalter_ausgeloest		: TON;
	fb_ton_temperatur_schaltschrank	: TON;
	fb_ton_ueberstrom_haspe			: TON;
	fb_ton_quitt						: TON;
	fb_ton_wz						: TON;
	fb_state_entry						: ST_StateEntry;
	sm_druckwaechter  				: BOOL := FALSE;
	sm_druckwaechter_hublift_links		: BOOL := FALSE;
	sm_schaltschrank 					: BOOL := FALSE;
	sm_ls_schalter 					: BOOL := FALSE;
	sm_haube_offen 					: BOOL := FALSE;
	sm_ueberstrom_haspel			: BOOL := FALSE;

	bm_schaltschrank 					: BOOL := FALSE;

	e_temperatur_schaltschrank 		AT %I* : BOOL;
	e_ls_schalter_ausgeloest 			AT %I* : BOOL;

	e_ueberstrom_haspel				AT %I* : BOOL;
	a_lampe_steuerung 				AT %Q* : BOOL;
	e_druckwaechter					AT %I* : BOOL;
	e_druckwaechter_hublift_links		AT %I* : BOOL;
	a_lampe_stoerung 				AT %Q* : BOOL;
	a_lampe_produktion 				AT %Q* : BOOL;
END_VAR
fb_tof_druck(IN:=e_druckwaechter , PT:= t#500ms, Q=> , ET=> );
fb_tof_druck_hublift_links(IN:=e_druckwaechter_hublift_links , PT:= t#500ms, Q=> , ET=> );
fb_ton_ls_schalter_ausgeloest(IN:=NOT e_ls_schalter_ausgeloest  , PT:= t#200ms, Q=> , ET=> );
fb_ton_temperatur_schaltschrank(IN:=NOT e_temperatur_schaltschrank  , PT:= t#200ms, Q=> , ET=> );
fb_ton_ueberstrom_haspe(IN:=NOT e_ueberstrom_haspel , PT:= t#200ms, Q=> , ET=> );

fb_ton_wz(IN:= , PT:= t#500ms, Q=> , ET=> );
fb_ton_quitt(IN:= , PT:= t#50ms, Q=> , ET=> );

a_lampe_steuerung := e_steuerung_ein ;
a_lampe_stoerung := b_lampe_stoerung;
a_lampe_produktion := b_lampe_produktion;

bm_schaltschrank:=fb_ton_temperatur_schaltschrank.Q;
ST_LampeMaterialMangel.b_materialmangel[4]:=bm_schaltschrank;

(*=======================Schrittkette=======================*)
fb_state_entry(
	i16_next_step:= ,
	i16_pos:= 1,
	s_debugtext:= ,
	E=> ,
	X=> ,
	i16_step=> ,
	i16_last_step=> );

CASE fb_state_entry.i16_step OF
(*=======================================================*)
	INIT_OBJ:
		IF st_config.b_config_fertig THEN
			fb_state_entry.i16_next_step := INIT;
		END_IF

(*=======================================================*)
	INIT:
		st_ctrl_out.b_fehler := FALSE;
		st_ctrl_out.b_bereit := FALSE;
		fb_ton_wz.IN := FALSE;
		fb_ton_quitt.IN := FALSE;
		sm_druckwaechter  := FALSE;
		sm_druckwaechter_hublift_links := FALSE;
		sm_schaltschrank  := FALSE;
		sm_ls_schalter  := FALSE;
		sm_haube_offen := FALSE;
		sm_ueberstrom_haspel := FALSE;
		bm_schaltschrank  := FALSE;
		(*-----------------------Weiterschaltbedingungen----------------------------*)
		fb_state_entry.i16_next_step := BEREIT;

(*=======================================================*)
	BEREIT:
		IF fb_state_entry.E THEN
			st_ctrl_out.b_bereit := TRUE;
		END_IF

		(*-----------------------Weiterschaltbedingungen----------------------------*)
		IF 	NOT fb_tof_druck.Q THEN
			sm_druckwaechter := TRUE;
			fb_state_entry.i16_next_step := FEHLER;
		END_IF
		IF	 fb_ton_ls_schalter_ausgeloest.Q THEN
			sm_ls_schalter := TRUE;
			fb_state_entry.i16_next_step := FEHLER;
		END_IF
		(*IF 	fb_ton_ueberstrom_foerderbaender.Q THEN
			sm_ueberstrom_foerderbaender := TRUE;
			fb_state_entry.i16_next_step := FEHLER;
		END_IF*)
		IF 	fb_ton_ueberstrom_haspe.Q THEN
			sm_ueberstrom_haspel := TRUE;
			fb_state_entry.i16_next_step := FEHLER;
		END_IF
		IF gst_datensatz.st_md.b_hublift_links_aktiv THEN
			IF NOT fb_tof_druck_hublift_links.Q THEN
				sm_druckwaechter_hublift_links := TRUE;
				fb_state_entry.i16_next_step := FEHLER;
			END_IF
		END_IF

(*		IF 	fb_ton_temperatur_schaltschrank.Q THEN
			sm_schaltschrank := TRUE;
			fb_state_entry.i16_next_step := FEHLER;
		END_IF*)

(*=======================================================*)
	FEHLER:
		IF fb_state_entry.E THEN
			st_ctrl_out.b_fehler := TRUE;
			fb_ton_quitt.IN := FALSE;
		END_IF

		(*-----------------------Weiterschaltbedingungen----------------------------*)
		IF st_ctrl_in.b_quitt AND NOT fb_state_entry.E THEN
			st_ctrl_out.b_fehler := FALSE;
			fb_ton_quitt.IN := TRUE;
		END_IF

		IF fb_ton_quitt.Q THEN
			fb_ton_quitt.IN := FALSE;
			fb_state_entry.i16_next_step := INIT;
		END_IF
END_CASE

fb_state_entry(
	i16_next_step:= , 
	i16_pos:= 2,
	s_debugtext:= ,
	E=> ,
	X=> ,
	i16_step=> ,
	i16_last_step=> );

IF st_config.b_config_fertig THEN
	(* Fehlermeldungen und Betriebsmeldungen ab dem Startindex in die globalen Meldungsarrays schreiben *)
	garr_stoermeldungen[st_config.i16_meld_startindex + 0] := FALSE;;
	garr_stoermeldungen[st_config.i16_meld_startindex + 1] := sm_druckwaechter;
	garr_stoermeldungen[st_config.i16_meld_startindex + 2] := sm_schaltschrank;
	garr_stoermeldungen[st_config.i16_meld_startindex + 3] := sm_ls_schalter;
	garr_stoermeldungen[st_config.i16_meld_startindex + 4] := sm_haube_offen;
	garr_stoermeldungen[st_config.i16_meld_startindex + 5] := sm_ueberstrom_haspel;
	garr_stoermeldungen[st_config.i16_meld_startindex + 6] := sm_druckwaechter_hublift_links;
	garr_stoermeldungen[st_config.i16_meld_startindex + 7] := FALSE;
	garr_stoermeldungen[st_config.i16_meld_startindex + 8] := FALSE;
	garr_stoermeldungen[st_config.i16_meld_startindex + 9] := FALSE;
	garr_stoermeldungen[st_config.i16_meld_startindex + 10] := FALSE;
	garr_stoermeldungen[st_config.i16_meld_startindex + 11] := FALSE;
	garr_stoermeldungen[st_config.i16_meld_startindex + 12] := FALSE;
	garr_stoermeldungen[st_config.i16_meld_startindex + 13] := FALSE;
	garr_stoermeldungen[st_config.i16_meld_startindex + 14] := FALSE;
	garr_stoermeldungen[st_config.i16_meld_startindex + 15] := FALSE;
	garr_stoermeldungen[st_config.i16_meld_startindex + 16] := FALSE;
	garr_stoermeldungen[st_config.i16_meld_startindex + 17] := FALSE;
	garr_stoermeldungen[st_config.i16_meld_startindex + 18] := FALSE;
	garr_stoermeldungen[st_config.i16_meld_startindex + 19] := FALSE;
	
	(* Betriebsmeldungen *)
	garr_betriebsmeldungen[st_config.i16_meld_startindex + 0] := bm_schaltschrank;
	garr_betriebsmeldungen[st_config.i16_meld_startindex + 1] := FALSE;
	garr_betriebsmeldungen[st_config.i16_meld_startindex + 2] := FALSE;
	garr_betriebsmeldungen[st_config.i16_meld_startindex + 3] := FALSE;
	garr_betriebsmeldungen[st_config.i16_meld_startindex + 4] := FALSE;
	garr_betriebsmeldungen[st_config.i16_meld_startindex + 5] := FALSE;
	garr_betriebsmeldungen[st_config.i16_meld_startindex + 6] := FALSE;
	garr_betriebsmeldungen[st_config.i16_meld_startindex + 7] := FALSE;
	garr_betriebsmeldungen[st_config.i16_meld_startindex + 8] := FALSE;
	garr_betriebsmeldungen[st_config.i16_meld_startindex + 9] := FALSE;
	garr_betriebsmeldungen[st_config.i16_meld_startindex + 10] := FALSE;
	garr_betriebsmeldungen[st_config.i16_meld_startindex + 11] := FALSE;
	garr_betriebsmeldungen[st_config.i16_meld_startindex + 12] := FALSE;
	garr_betriebsmeldungen[st_config.i16_meld_startindex + 13] := FALSE;
	garr_betriebsmeldungen[st_config.i16_meld_startindex + 14] := FALSE;
	garr_betriebsmeldungen[st_config.i16_meld_startindex + 15] := FALSE;
	garr_betriebsmeldungen[st_config.i16_meld_startindex + 16] := FALSE;
	garr_betriebsmeldungen[st_config.i16_meld_startindex + 17] := FALSE;
	garr_betriebsmeldungen[st_config.i16_meld_startindex + 18] := FALSE;
	garr_betriebsmeldungen[st_config.i16_meld_startindex + 19] := FALSE;
END_IF
END_PROGRAM

(* POU Gemeinsamkeiten17xx/Haspel/Mehrfach/ST_Haspel_Kontroller_2H, ST *)
PROGRAM ST_Haspel_Kontroller_2H
VAR_INPUT
	t_abschaltzeit_motor			: TIME;
	b_drehrichtung_antrieb_links	: BOOL;
	st_config						: struct_config;
	e_druckwaechter				: BOOL;
	e_steuerung_ein				: BOOL;
	st_ctrl_in						: struct_ctrl_in;
	haspel1_ctrl_in				: struct_ctrl_out;
	haspel2_ctrl_in				: struct_ctrl_out;
END_VAR
VAR_IN_OUT
	st_visu						: struct_visu;
END_VAR
VAR_OUTPUT
	st_ctrl_out					: struct_ctrl_out;
	haspel1_ctrl_out				: struct_ctrl_in;
	haspel2_ctrl_out				: struct_ctrl_in;
	b_materialmangel_bandende	: BOOL := FALSE;
END_VAR
VAR
	fb_ton_wz					: TON;
	fb_ton_uez					: TON;
	fb_ton_vz					: TON;
	fb_tof_motor					: TOF;
	fb_ton_quitt					: TON;
	fb_r_trig_start					: R_TRIG;
	fb_state_entry					: ST_StateEntry;
	sm_haspel_nicht_bb			: BOOL := FALSE;
	e_haspelmotor_bb			AT %I* : BOOL;
	a_motor_drehrichtung_rechts	AT %Q* : BOOL;
	a_motor_drehrichtung_links		AT %Q* : BOOL;
END_VAR
(* Zeiten *)
fb_ton_wz(IN:= , PT:= , Q=>  , ET=> );
fb_ton_uez(IN:= , PT:= , Q=>  , ET=> );
fb_ton_vz(IN:= , PT:= , Q=>  , ET=> );
fb_tof_motor(IN:= , PT:= t_abschaltzeit_motor, Q=> , ET=> );
fb_ton_quitt(IN:= , PT:= t#100ms, Q=> , ET=> );

(* Flanken *)
fb_r_trig_start(CLK:= st_ctrl_in.b_start, Q=> );

(* Haspelmotor *)
IF 	e_steuerung_ein AND
	e_druckwaechter AND
	fb_tof_motor.Q AND
	fb_state_entry.i16_next_step <> FEHLER THEN
		a_motor_drehrichtung_links 	:= b_drehrichtung_antrieb_links;
		a_motor_drehrichtung_rechts := NOT b_drehrichtung_antrieb_links;
ELSE
	a_motor_drehrichtung_links 	:= FALSE;
	a_motor_drehrichtung_rechts := FALSE;
END_IF

(* Freigabe für die jeweils benutzte Haspel setzen. Wird für Bandende benötigt (ST_Haspel_V2)*)
CASE gst_datensatz.st_md.i16_typ_zelle OF

KEINE_ZELLE:
		;

BESTUECKZELLE_1700:
	IF zyl_bandeinzuege_verschieben.st_ctrl.out.b_ausgefahren THEN
		haspel1_ctrl_out.b_freigabe := TRUE;
		haspel2_ctrl_out.b_freigabe := FALSE;
	ELSIF zyl_bandeinzuege_verschieben.st_ctrl.out.b_eingefahren THEN
		haspel1_ctrl_out.b_freigabe := FALSE;
		haspel2_ctrl_out.b_freigabe := TRUE;
	END_IF

RASTERFOLIE:
	haspel1_ctrl_out.b_freigabe := TRUE;
	haspel2_ctrl_out.b_freigabe := FALSE;

BESTUECKZELLE_1720:
	haspel1_ctrl_out.b_freigabe := TRUE;
	haspel2_ctrl_out.b_freigabe := TRUE;

END_CASE

(* Bandende von Haspel rechts bzw. links *)
IF	(gi16_betriebsart = AUTO OR gi16_betriebsart = TIPPEN) AND
	(haspel1_ctrl_in.b_bandende OR haspel2_ctrl_in.b_bandende )
	THEN
		st_ctrl_out.b_bandende := b_materialmangel_bandende := TRUE;
ELSE
		st_ctrl_out.b_bandende := b_materialmangel_bandende := FALSE;
END_IF

(* Toplevel *)
IF fb_state_entry.i16_next_step > INIT AND fb_state_entry.i16_next_step < FEHLER THEN
	IF fb_state_entry.i16_next_step < STOP THEN
		IF st_ctrl_in.b_stop THEN
			fb_state_entry.i16_next_step := STOP;
		END_IF
	END_IF
	(* Allgemeine Fehler *)
	IF haspel1_ctrl_in.b_fehler OR haspel2_ctrl_in.b_fehler THEN
		fb_state_entry.i16_next_step := FEHLER;
	END_IF
END_IF


(* ======================================Schrittkette======================================== *)
fb_state_entry(
	i16_next_step:= ,
	i16_pos:= 1,
	s_debugtext:= ,
	E=> ,
	X=> , 
	i16_step=> ,
	i16_last_step=> );

CASE fb_state_entry.i16_step OF
(*=======================================================*)
	INIT_OBJ:
		IF st_config.b_config_fertig THEN
			fb_state_entry.i16_next_step := INIT;
		END_IF

(*=======================================================*)
	INIT:
		IF fb_state_entry.E THEN
			fb_ton_wz.IN := FALSE;
			fb_ton_uez.IN	:= FALSE;
			fb_ton_vz.IN := FALSE;
			fb_ton_quitt.IN := FALSE;
			a_motor_drehrichtung_links := FALSE;
			a_motor_drehrichtung_rechts := FALSE;
			sm_haspel_nicht_bb := FALSE;
			st_ctrl_out.b_fehler := FALSE;
			st_ctrl_out.b_bereit := FALSE;
			st_ctrl_out.b_fertig := FALSE;
			haspel1_ctrl_out.b_stop := FALSE;
			haspel2_ctrl_out.b_stop := FALSE;
			haspel1_ctrl_out.b_init := FALSE;
			haspel2_ctrl_out.b_init := FALSE;
		END_IF

		(*-----------------------Weiterschaltbedingungen----------------------------*)
		IF st_ctrl_in.b_init THEN
			haspel1_ctrl_out.b_quitt := FALSE;
			haspel2_ctrl_out.b_quitt := FALSE;
			fb_state_entry.i16_next_step :=20;
		END_IF

(*=======================================================*)
	20:	(* Haspeln initialisieren *)
		IF fb_state_entry.E THEN
			haspel1_ctrl_out.b_init := TRUE;
			haspel2_ctrl_out.b_init := TRUE;
		END_IF

		(*-----------------------Weiterschaltbedingungen----------------------------*)
		IF  haspel1_ctrl_in.b_bereit AND haspel2_ctrl_in.b_bereit THEN
			haspel1_ctrl_out.b_init := FALSE;
			haspel2_ctrl_out.b_init := FALSE;
			fb_tof_motor.IN := TRUE;
			fb_state_entry.i16_next_step := BEREIT;
		END_IF

(*=======================================================*)
	BEREIT: (* Haspelmotor läuft *)
		IF fb_state_entry.E THEN
			st_ctrl_out.b_bereit := TRUE;
			st_ctrl_out.b_fertig := TRUE;
		END_IF

		IF haspel1_ctrl_in.b_kontroller_start OR haspel2_ctrl_in.b_kontroller_start THEN	(* Abschaltzeit für Haspelmotor nachtriggern*)
			fb_tof_motor.IN := TRUE;
		ELSE
			fb_tof_motor.IN := FALSE;
		END_IF

(*=======================================================*)
	FEHLER:
		IF fb_state_entry.E THEN
			st_ctrl_out.b_fehler := TRUE;
			fb_tof_motor.IN := FALSE;
			haspel1_ctrl_out.b_quitt := FALSE;
			haspel2_ctrl_out.b_quitt := FALSE;
			haspel1_ctrl_out.b_stop := FALSE;
			haspel2_ctrl_out.b_stop := FALSE;
			fb_ton_quitt.IN := FALSE;
		END_IF

		(*-----------------------Weiterschaltbedingungen----------------------------*)
		IF st_ctrl_in.b_quitt AND NOT fb_state_entry.E THEN
			haspel1_ctrl_out.b_quitt := TRUE;
			haspel2_ctrl_out.b_quitt := TRUE;
			st_ctrl_out.b_fehler := FALSE;
			fb_ton_quitt.IN := TRUE;
		END_IF

		IF fb_ton_quitt.Q THEN
			fb_ton_quitt.IN := FALSE;
			fb_state_entry.i16_next_step := INIT;
		END_IF

(*=======================================================*)
	STOP:
		IF fb_state_entry.E THEN
			fb_tof_motor.IN := FALSE;
			haspel1_ctrl_out.b_stop := TRUE;
			haspel2_ctrl_out.b_stop := TRUE;
			haspel1_ctrl_out.b_quitt := FALSE;
			haspel2_ctrl_out.b_quitt := FALSE;
			fb_ton_quitt.IN := FALSE;
		END_IF

		(*-----------------------Weiterschaltbedingungen----------------------------*)
		IF st_ctrl_in.b_quitt AND NOT fb_state_entry.E THEN
			haspel1_ctrl_out.b_stop := FALSE;
			haspel2_ctrl_out.b_stop := FALSE;
			haspel1_ctrl_out.b_quitt := TRUE;
			haspel2_ctrl_out.b_quitt := TRUE;
			fb_ton_quitt.IN := TRUE;
		END_IF

		IF fb_ton_quitt.Q THEN
			fb_ton_quitt.IN := FALSE;
			fb_state_entry.i16_next_step := INIT;
		END_IF
END_CASE

fb_state_entry(
	i16_next_step:= , 
	i16_pos:= 2,
	s_debugtext:= ,
	E=> , 
	X=> , 
	i16_step=> ,
	i16_last_step=> );

IF st_config.b_config_fertig THEN
	(* Fehlermeldungen und Betriebsmeldungen ab dem Startindex in die globalen Meldungsarrays schreiben *)
	garr_stoermeldungen[st_config.i16_meld_startindex + 0] := sm_haspel_nicht_bb;
	garr_stoermeldungen[st_config.i16_meld_startindex + 1] := FALSE;
	garr_stoermeldungen[st_config.i16_meld_startindex + 2] := FALSE;
	garr_stoermeldungen[st_config.i16_meld_startindex + 3] := FALSE;
	garr_stoermeldungen[st_config.i16_meld_startindex + 4] := FALSE;
	garr_stoermeldungen[st_config.i16_meld_startindex + 5] := FALSE;
	garr_stoermeldungen[st_config.i16_meld_startindex + 6] := FALSE;
	garr_stoermeldungen[st_config.i16_meld_startindex + 7] := FALSE;
	garr_stoermeldungen[st_config.i16_meld_startindex + 8] := FALSE;
	garr_stoermeldungen[st_config.i16_meld_startindex + 9] := FALSE;
	garr_stoermeldungen[st_config.i16_meld_startindex + 10] := FALSE;
	garr_stoermeldungen[st_config.i16_meld_startindex + 11] := FALSE;
	garr_stoermeldungen[st_config.i16_meld_startindex + 12] := FALSE;
	garr_stoermeldungen[st_config.i16_meld_startindex + 13] := FALSE;
	garr_stoermeldungen[st_config.i16_meld_startindex + 14] := FALSE;
	garr_stoermeldungen[st_config.i16_meld_startindex + 15] := FALSE;
	garr_stoermeldungen[st_config.i16_meld_startindex + 16] := FALSE;
	garr_stoermeldungen[st_config.i16_meld_startindex + 17] := FALSE;
	garr_stoermeldungen[st_config.i16_meld_startindex + 18] := FALSE;
	garr_stoermeldungen[st_config.i16_meld_startindex + 19] := FALSE;
	
	garr_betriebsmeldungen[st_config.i16_meld_startindex + 0] := FALSE;
	garr_betriebsmeldungen[st_config.i16_meld_startindex + 1] := FALSE;
	garr_betriebsmeldungen[st_config.i16_meld_startindex + 2] := FALSE;
	garr_betriebsmeldungen[st_config.i16_meld_startindex + 3] := FALSE;
	garr_betriebsmeldungen[st_config.i16_meld_startindex + 4] := FALSE;
	garr_betriebsmeldungen[st_config.i16_meld_startindex + 5] := FALSE;
	garr_betriebsmeldungen[st_config.i16_meld_startindex + 6] := FALSE;
	garr_betriebsmeldungen[st_config.i16_meld_startindex + 7] := FALSE;
	garr_betriebsmeldungen[st_config.i16_meld_startindex + 8] := FALSE;
	garr_betriebsmeldungen[st_config.i16_meld_startindex + 9] := FALSE;
	garr_betriebsmeldungen[st_config.i16_meld_startindex + 10] := FALSE;
	garr_betriebsmeldungen[st_config.i16_meld_startindex + 11] := FALSE;
	garr_betriebsmeldungen[st_config.i16_meld_startindex + 12] := FALSE;
	garr_betriebsmeldungen[st_config.i16_meld_startindex + 13] := FALSE;
	garr_betriebsmeldungen[st_config.i16_meld_startindex + 14] := FALSE;
	garr_betriebsmeldungen[st_config.i16_meld_startindex + 15] := FALSE;
	garr_betriebsmeldungen[st_config.i16_meld_startindex + 16] := FALSE;
	garr_betriebsmeldungen[st_config.i16_meld_startindex + 17] := FALSE;
	garr_betriebsmeldungen[st_config.i16_meld_startindex + 18] := FALSE;
	garr_betriebsmeldungen[st_config.i16_meld_startindex + 19] := FALSE;
END_IF
END_PROGRAM

(* POU Gemeinsamkeiten17xx/Haspel/Mehrfach/ST_Haspel_Kontroller_4H, ST *)
PROGRAM ST_Haspel_Kontroller_4H
VAR_INPUT
	t_abschaltzeit_motor			: TIME;
	b_drehrichtung_antrieb_links	: BOOL;
	st_config						: struct_config;
	e_druckwaechter				: BOOL;
	e_steuerung_ein				: BOOL;
	st_ctrl_in						: struct_ctrl_in;
	haspel1_ctrl_in				: struct_ctrl_out;
	haspel2_ctrl_in				: struct_ctrl_out;
	haspel3_ctrl_in				: struct_ctrl_out;
	haspel4_ctrl_in				: struct_ctrl_out;
END_VAR
VAR_IN_OUT
	st_visu						: struct_visu;
END_VAR
VAR_OUTPUT
	st_ctrl_out					: struct_ctrl_out;
	haspel1_ctrl_out				: struct_ctrl_in;
	haspel2_ctrl_out				: struct_ctrl_in;
	haspel3_ctrl_out				: struct_ctrl_in;
	haspel4_ctrl_out				: struct_ctrl_in;
END_VAR
VAR
	fb_ton_wz					: TON;
	fb_ton_uez					: TON;
	fb_ton_vz					: TON;
	fb_ton_quitt					: TON;
	fb_tof_motor					: TOF;
	b_motor_laeuft				: BOOL := FALSE;
	fb_state_entry					: ST_StateEntry;
	a_motor_drehrichtung_rechts	AT %Q* : BOOL;
	a_motor_drehrichtung_links		AT %Q* : BOOL;
END_VAR
(* Zeiten *)
fb_ton_wz(IN:= , PT:= , Q=>  , ET=> );
fb_ton_uez(IN:= , PT:= , Q=>  , ET=> );
fb_ton_vz(IN:= , PT:= , Q=>  , ET=> );
fb_tof_motor(IN:= , PT:= t_abschaltzeit_motor, Q=> , ET=> );
fb_ton_quitt(IN:= , PT:= t#100ms, Q=> , ET=> );

b_motor_laeuft := a_motor_drehrichtung_links OR a_motor_drehrichtung_rechts;

(* Bandende von Haspel rechts bzw. links *)
IF	(gi16_betriebsart = AUTO OR gi16_betriebsart = TIPPEN) AND
 	(haspel1_ctrl_in.b_bandende OR
	haspel2_ctrl_in.b_bandende OR
	haspel3_ctrl_in.b_bandende OR
	haspel4_ctrl_in.b_bandende)
	THEN
		st_ctrl_out.b_bandende := TRUE;
ELSE
		st_ctrl_out.b_bandende := FALSE;
END_IF

(* Toplevel *)
IF fb_state_entry.i16_next_step > INIT AND fb_state_entry.i16_next_step < FEHLER THEN
	IF fb_state_entry.i16_next_step < STOP THEN
		IF st_ctrl_in.b_stop THEN
			fb_state_entry.i16_next_step := STOP;
		END_IF
	END_IF
	IF 	haspel1_ctrl_in.b_fehler OR
		haspel2_ctrl_in.b_fehler OR
		haspel3_ctrl_in.b_fehler OR
		haspel4_ctrl_in.b_fehler
		THEN
			fb_state_entry.i16_next_step := FEHLER;
	END_IF
END_IF

(* ==================================Schrittkette================================ *)
fb_state_entry(
	i16_next_step:= , 
	i16_pos:= 1,
	s_debugtext:= ,
	E=> ,
	X=> , 
	i16_step=> ,
	i16_last_step=> );

CASE fb_state_entry.i16_step OF
(*=======================================================*)
	INIT_OBJ:
		IF st_config.b_config_fertig THEN
			fb_state_entry.i16_next_step := INIT;
		END_IF

(*=======================================================*)
	INIT:
		IF fb_state_entry.E THEN
			fb_ton_wz.IN := FALSE;
			fb_ton_uez.IN	:= FALSE;
			fb_ton_vz.IN := FALSE;
			fb_ton_quitt.IN := FALSE;
			a_motor_drehrichtung_links 	:= FALSE;
			a_motor_drehrichtung_rechts := FALSE;
			st_ctrl_out.b_fehler := FALSE;
			st_ctrl_out.b_bereit := FALSE;
			st_ctrl_out.b_fertig := FALSE;
			haspel1_ctrl_out.b_init := FALSE;
			haspel2_ctrl_out.b_init := FALSE;
			haspel3_ctrl_out.b_init := FALSE;
			haspel4_ctrl_out.b_init := FALSE;
		END_IF

		(*-----------------------Weiterschaltbedingungen----------------------------*)
		IF st_ctrl_in.b_init THEN
			haspel1_ctrl_out.b_quitt := FALSE;
			haspel2_ctrl_out.b_quitt := FALSE;
			haspel3_ctrl_out.b_quitt := FALSE;
			haspel4_ctrl_out.b_quitt := FALSE;
			fb_state_entry.i16_next_step :=20;
		END_IF

(*=======================================================*)
	20:
		IF fb_state_entry.E THEN
			haspel1_ctrl_out.b_init := TRUE;
			haspel2_ctrl_out.b_init := TRUE;
			haspel3_ctrl_out.b_init := TRUE;
			haspel4_ctrl_out.b_init := TRUE;
		END_IF
		(*-----------------------Weiterschaltbedingungen----------------------------*)
		IF  	haspel1_ctrl_in.b_bereit AND
			haspel2_ctrl_in.b_bereit AND
			haspel3_ctrl_in.b_bereit AND
			haspel4_ctrl_in.b_bereit
			THEN
				haspel1_ctrl_out.b_init := FALSE;
				haspel2_ctrl_out.b_init := FALSE;
				haspel3_ctrl_out.b_init := FALSE;
				haspel4_ctrl_out.b_init := FALSE;
				fb_tof_motor.IN := TRUE;
				fb_state_entry.i16_next_step := BEREIT;
		END_IF

(*=======================================================*)
	BEREIT: (* Haspelmotor läuft *)
		IF fb_state_entry.E THEN
			st_ctrl_out.b_bereit := TRUE;
		END_IF

		a_motor_drehrichtung_links 	:= e_druckwaechter AND fb_tof_motor.Q AND b_drehrichtung_antrieb_links;
		a_motor_drehrichtung_rechts := e_druckwaechter AND fb_tof_motor.Q AND NOT b_drehrichtung_antrieb_links;

		(* Abschaltzeit für Haspelmotor nachtriggern*)
		IF 	haspel1_ctrl_in.b_kontroller_start OR
			haspel2_ctrl_in.b_kontroller_start OR
			haspel3_ctrl_in.b_kontroller_start OR
			haspel4_ctrl_in.b_kontroller_start
			THEN
				fb_tof_motor.IN := TRUE;
		ELSE
			fb_tof_motor.IN := FALSE;
		END_IF

(*=======================================================*)
	FEHLER:
		IF fb_state_entry.E THEN
			fb_ton_quitt.IN := FALSE;
			st_ctrl_out.b_fehler := TRUE;
			haspel1_ctrl_out.b_stop := FALSE;
			haspel2_ctrl_out.b_stop := FALSE;
			haspel3_ctrl_out.b_stop := FALSE;
			haspel4_ctrl_out.b_stop := FALSE;
			haspel1_ctrl_out.b_quitt := FALSE;
			haspel2_ctrl_out.b_quitt := FALSE;
			haspel3_ctrl_out.b_quitt := FALSE;
			haspel4_ctrl_out.b_quitt := FALSE;
			a_motor_drehrichtung_links 	:= FALSE;
			a_motor_drehrichtung_rechts := FALSE;
		END_IF

		(*-----------------------Weiterschaltbedingungen----------------------------*)
		IF st_ctrl_in.b_quitt AND NOT fb_state_entry.E THEN
			haspel1_ctrl_out.b_quitt := TRUE;
			haspel2_ctrl_out.b_quitt := TRUE;
			haspel3_ctrl_out.b_quitt := TRUE;
			haspel4_ctrl_out.b_quitt := TRUE;
			st_ctrl_out.b_fehler := FALSE;
			fb_ton_quitt.IN := TRUE;
		END_IF

		IF fb_ton_quitt.Q THEN
			fb_ton_quitt.IN := FALSE;
			fb_state_entry.i16_next_step := INIT;
		END_IF

(*=======================================================*)
	STOP:
		IF fb_state_entry.E THEN
			a_motor_drehrichtung_links 	:= FALSE;
			a_motor_drehrichtung_rechts := FALSE;
			haspel1_ctrl_out.b_stop := TRUE;
			haspel2_ctrl_out.b_stop := TRUE;
			haspel3_ctrl_out.b_stop := TRUE;
			haspel4_ctrl_out.b_stop := TRUE;
			haspel1_ctrl_out.b_quitt := FALSE;
			haspel2_ctrl_out.b_quitt := FALSE;
			haspel3_ctrl_out.b_quitt := FALSE;
			haspel4_ctrl_out.b_quitt := FALSE;
			fb_ton_quitt.IN := FALSE;
		END_IF

		(*-----------------------Weiterschaltbedingungen----------------------------*)
		IF st_ctrl_in.b_quitt AND NOT fb_state_entry.E THEN
			haspel1_ctrl_out.b_stop := FALSE;
			haspel2_ctrl_out.b_stop := FALSE;
			haspel3_ctrl_out.b_stop := FALSE;
			haspel4_ctrl_out.b_stop := FALSE;
			haspel1_ctrl_out.b_quitt := TRUE;
			haspel2_ctrl_out.b_quitt := TRUE;
			haspel3_ctrl_out.b_quitt := TRUE;
			haspel4_ctrl_out.b_quitt := TRUE;

			fb_ton_quitt.IN := TRUE;
		END_IF

		IF fb_ton_quitt.Q THEN
			fb_ton_quitt.IN := FALSE;
			fb_state_entry.i16_next_step := INIT;
		END_IF
END_CASE

fb_state_entry(
	i16_next_step:= , 
	i16_pos:= 2,
	s_debugtext:= ,
	E=> , 
	X=> , 
	i16_step=> ,
	i16_last_step=> );

IF st_config.b_config_fertig THEN
	(* Fehlermeldungen und Betriebsmeldungen ab dem Startindex in die globalen Meldungsarrays schreiben *)
	garr_stoermeldungen[st_config.i16_meld_startindex + 0] := FALSE;
	garr_stoermeldungen[st_config.i16_meld_startindex + 1] := FALSE;
	garr_stoermeldungen[st_config.i16_meld_startindex + 2] := FALSE;
	garr_stoermeldungen[st_config.i16_meld_startindex + 3] := FALSE;
	garr_stoermeldungen[st_config.i16_meld_startindex + 4] := FALSE;
	garr_stoermeldungen[st_config.i16_meld_startindex + 5] := FALSE;
	garr_stoermeldungen[st_config.i16_meld_startindex + 6] := FALSE;
	garr_stoermeldungen[st_config.i16_meld_startindex + 7] := FALSE;
	garr_stoermeldungen[st_config.i16_meld_startindex + 8] := FALSE;
	garr_stoermeldungen[st_config.i16_meld_startindex + 9] := FALSE;
	garr_stoermeldungen[st_config.i16_meld_startindex + 10] := FALSE;
	garr_stoermeldungen[st_config.i16_meld_startindex + 11] := FALSE;
	garr_stoermeldungen[st_config.i16_meld_startindex + 12] := FALSE;
	garr_stoermeldungen[st_config.i16_meld_startindex + 13] := FALSE;
	garr_stoermeldungen[st_config.i16_meld_startindex + 14] := FALSE;
	garr_stoermeldungen[st_config.i16_meld_startindex + 15] := FALSE;
	garr_stoermeldungen[st_config.i16_meld_startindex + 16] := FALSE;
	garr_stoermeldungen[st_config.i16_meld_startindex + 17] := FALSE;
	garr_stoermeldungen[st_config.i16_meld_startindex + 18] := FALSE;
	garr_stoermeldungen[st_config.i16_meld_startindex + 19] := FALSE;
	
	garr_betriebsmeldungen[st_config.i16_meld_startindex + 0] := FALSE;
	garr_betriebsmeldungen[st_config.i16_meld_startindex + 1] := FALSE;
	garr_betriebsmeldungen[st_config.i16_meld_startindex + 2] := FALSE;
	garr_betriebsmeldungen[st_config.i16_meld_startindex + 3] := FALSE;
	garr_betriebsmeldungen[st_config.i16_meld_startindex + 4] := FALSE;
	garr_betriebsmeldungen[st_config.i16_meld_startindex + 5] := FALSE;
	garr_betriebsmeldungen[st_config.i16_meld_startindex + 6] := FALSE;
	garr_betriebsmeldungen[st_config.i16_meld_startindex + 7] := FALSE;
	garr_betriebsmeldungen[st_config.i16_meld_startindex + 8] := FALSE;
	garr_betriebsmeldungen[st_config.i16_meld_startindex + 9] := FALSE;
	garr_betriebsmeldungen[st_config.i16_meld_startindex + 10] := FALSE;
	garr_betriebsmeldungen[st_config.i16_meld_startindex + 11] := FALSE;
	garr_betriebsmeldungen[st_config.i16_meld_startindex + 12] := FALSE;
	garr_betriebsmeldungen[st_config.i16_meld_startindex + 13] := FALSE;
	garr_betriebsmeldungen[st_config.i16_meld_startindex + 14] := FALSE;
	garr_betriebsmeldungen[st_config.i16_meld_startindex + 15] := FALSE;
	garr_betriebsmeldungen[st_config.i16_meld_startindex + 16] := FALSE;
	garr_betriebsmeldungen[st_config.i16_meld_startindex + 17] := FALSE;
	garr_betriebsmeldungen[st_config.i16_meld_startindex + 18] := FALSE;
	garr_betriebsmeldungen[st_config.i16_meld_startindex + 19] := FALSE;
END_IF
END_PROGRAM

(* POU Gemeinsamkeiten17xx/Initialisierung/Startup/ST_Datainit_Achsen, ST *)
PROGRAM ST_Datainit_Achsen
VAR
	b_config_fertig			: BOOL := FALSE;
END_VAR
IF	NOT axis_bestueckachse.st_config.b_config_fertig OR
	NOT axis_virt_master.st_config.b_config_fertig OR
	NOT axis_z_achse.st_config.b_config_fertig OR
	NOT axis_y_achse.st_config.b_config_fertig OR
	NOT axis_bandeinzug_achse.st_config.b_config_fertig OR
	NOT axis_transport_wt_achse.st_config.b_config_fertig
	THEN
		CASE gst_datensatz.st_md.i16_typ_zelle OF
			KEINE_ZELLE:
				;
			BESTUECKZELLE_1700:
				(* Virtuelle Masterachse *)
				axis_virt_master.st_config.b_config_fertig := FALSE;
				axis_virt_master.st_config.b_limitsensor_negativ_vorhanden := FALSE;
				axis_virt_master.st_config.b_limitsensor_positiv_vorhanden := FALSE;
				axis_virt_master.st_config.b_refsensor_vorhanden := FALSE;
				axis_virt_master.st_config.r_getriebefaktor := 1.0;
				axis_virt_master.st_config.i16_achstyp := RUND_VIRTUELL;
				axis_virt_master.st_config.i16_meld_startindex := 1400;
				axis_virt_master.st_config.s_beschreibung := ' ';
				axis_virt_master.st_config.s_instanz_name := 'Virtuelle Masterachse';
				axis_virt_master.st_config.ui16_ethercat_slave_id := 0;
				axis_virt_master.st_config.ui16_ethercat_adr := 0;
				axis_virt_master.st_config.b_config_fertig := TRUE;
				(* Bestueckachse *)
				axis_bestueckachse.st_config.b_config_fertig := FALSE;
				axis_bestueckachse.st_config.b_limitsensor_negativ_vorhanden := FALSE;
				axis_bestueckachse.st_config.b_limitsensor_positiv_vorhanden := FALSE;
				axis_bestueckachse.st_config.b_refsensor_vorhanden := FALSE;
				axis_bestueckachse.st_config.r_getriebefaktor := 1.0;
				axis_bestueckachse.st_config.i16_achstyp := RUND;
				axis_bestueckachse.st_config.i16_meld_startindex := 1000;
				axis_bestueckachse.st_config.s_beschreibung := ' ';
				axis_bestueckachse.st_config.s_instanz_name := 'Bestückachse';
				axis_bestueckachse.st_config.ui16_ethercat_slave_id := 42;
				axis_bestueckachse.st_config.ui16_ethercat_adr := 1024;
				axis_bestueckachse.st_config.b_config_fertig := TRUE;
				(* Servobandeinzug *)
				axis_bandeinzug_achse.st_config.b_config_fertig := FALSE;
				axis_bandeinzug_achse.st_config.b_limitsensor_negativ_vorhanden := FALSE;
				axis_bandeinzug_achse.st_config.b_limitsensor_positiv_vorhanden := FALSE;
				axis_bandeinzug_achse.st_config.b_refsensor_vorhanden := FALSE;
				axis_bandeinzug_achse.st_config.r_getriebefaktor := 1.0;
				axis_bandeinzug_achse.st_config.i16_achstyp := RUND;
				axis_bandeinzug_achse.st_config.i16_meld_startindex := 1300;
				axis_bandeinzug_achse.st_config.s_beschreibung := ' ';
				axis_bandeinzug_achse.st_config.s_instanz_name := 'Servobandeinzug';
				axis_bandeinzug_achse.st_config.ui16_ethercat_slave_id := 42;
				axis_bandeinzug_achse.st_config.ui16_ethercat_adr := 1024;
				(* Z-Achse *)
				axis_z_achse.st_config.b_config_fertig := FALSE;
				axis_z_achse.st_config.b_limitsensor_negativ_vorhanden := FALSE;
				axis_z_achse.st_config.b_limitsensor_positiv_vorhanden := FALSE;
				axis_z_achse.st_config.b_refsensor_vorhanden := FALSE;
				axis_z_achse.st_config.r_getriebefaktor := 1.0;
				axis_z_achse.st_config.i16_achstyp := LINEAR;
				axis_z_achse.st_config.i16_meld_startindex := 1100;
				axis_z_achse.st_config.s_beschreibung := ' ';
				axis_z_achse.st_config.s_instanz_name := 'Z-Achse';
				axis_z_achse.st_config.ui16_ethercat_slave_id := 43;
				axis_z_achse.st_config.ui16_ethercat_adr := 1026;
				axis_z_achse.st_config.b_config_fertig := TRUE;
				(* Y-Achse *)
				axis_y_achse.st_config.b_config_fertig := FALSE;
				axis_y_achse.st_config.b_limitsensor_negativ_vorhanden := FALSE;
				axis_y_achse.st_config.b_limitsensor_positiv_vorhanden := FALSE;
				axis_y_achse.st_config.b_refsensor_vorhanden := FALSE;
				axis_y_achse.st_config.r_getriebefaktor := 1.0;
				axis_y_achse.st_config.i16_achstyp := LINEAR;
				axis_y_achse.st_config.i16_meld_startindex := 1200;
				axis_y_achse.st_config.s_beschreibung := ' ';
				axis_y_achse.st_config.s_instanz_name := 'Y-Achse';
				axis_y_achse.st_config.ui16_ethercat_slave_id := 43;
				axis_y_achse.st_config.ui16_ethercat_adr := 1026;
				axis_y_achse.st_config.b_config_fertig := TRUE;
				(* Transport WT Achse *)
				axis_transport_wt_achse.st_config.b_config_fertig := FALSE;
				axis_transport_wt_achse.st_config.b_limitsensor_negativ_vorhanden := FALSE;
				axis_transport_wt_achse.st_config.b_limitsensor_positiv_vorhanden := FALSE;
				axis_transport_wt_achse.st_config.b_refsensor_vorhanden := FALSE;
				axis_transport_wt_achse.st_config.r_getriebefaktor := 1.0;
				axis_transport_wt_achse.st_config.i16_achstyp := LINEAR;
				axis_transport_wt_achse.st_config.i16_meld_startindex := 1500;
				axis_transport_wt_achse.st_config.s_beschreibung := ' ';
				axis_transport_wt_achse.st_config.s_instanz_name := 'Transport_WT_Achse';
				axis_transport_wt_achse.st_config.ui16_ethercat_slave_id :=43;
				axis_transport_wt_achse.st_config.ui16_ethercat_adr :=1026;
				axis_transport_wt_achse.st_config.b_config_fertig := TRUE;

				axis_bandeinzug_achse.st_config.b_config_fertig := TRUE;

			BESTUECKZELLE_1720:
				(* Virtuelle Masterachse *)
				axis_virt_master.st_config.b_config_fertig := FALSE;
				axis_virt_master.st_config.b_limitsensor_negativ_vorhanden := FALSE;
				axis_virt_master.st_config.b_limitsensor_positiv_vorhanden := FALSE;
				axis_virt_master.st_config.b_refsensor_vorhanden := FALSE;
				axis_virt_master.st_config.r_getriebefaktor := 1.0;
				axis_virt_master.st_config.i16_achstyp := RUND_VIRTUELL;
				axis_virt_master.st_config.i16_meld_startindex := 1400;
				axis_virt_master.st_config.s_beschreibung := ' ';
				axis_virt_master.st_config.s_instanz_name := 'Virtuelle Masterachse';
				axis_virt_master.st_config.ui16_ethercat_slave_id := 0;
				axis_virt_master.st_config.ui16_ethercat_adr := 0;
				axis_virt_master.st_config.b_config_fertig := TRUE;
				(* Bestueckachse *)
				axis_bestueckachse.st_config.b_config_fertig := FALSE;
				axis_bestueckachse.st_config.b_limitsensor_negativ_vorhanden := FALSE;
				axis_bestueckachse.st_config.b_limitsensor_positiv_vorhanden := FALSE;
				axis_bestueckachse.st_config.b_refsensor_vorhanden := FALSE;
				axis_bestueckachse.st_config.r_getriebefaktor := 1.0;
				axis_bestueckachse.st_config.i16_achstyp := RUND;
				axis_bestueckachse.st_config.i16_meld_startindex := 1000;
				axis_bestueckachse.st_config.s_beschreibung := ' ';
				axis_bestueckachse.st_config.s_instanz_name := 'Bestückachse';
				axis_bestueckachse.st_config.ui16_ethercat_slave_id := 40;
				axis_bestueckachse.st_config.ui16_ethercat_adr := 1010;
				axis_bestueckachse.st_config.b_config_fertig := TRUE;
				(* Z-Achse *)
				axis_z_achse.st_config.b_config_fertig := FALSE;
				axis_z_achse.st_config.b_limitsensor_negativ_vorhanden := TRUE;
				axis_z_achse.st_config.b_limitsensor_positiv_vorhanden := TRUE;
				axis_z_achse.st_config.b_refsensor_vorhanden := FALSE;
				axis_z_achse.st_config.r_getriebefaktor := 1.0;
				axis_z_achse.st_config.i16_achstyp := LINEAR;
				axis_z_achse.st_config.i16_meld_startindex := 1100;
				axis_z_achse.st_config.s_beschreibung := ' ';
				axis_z_achse.st_config.s_instanz_name := 'Z-Achse';
				axis_z_achse.st_config.ui16_ethercat_slave_id := 7;
				axis_z_achse.st_config.ui16_ethercat_adr := 1012;
				axis_z_achse.st_config.b_config_fertig := TRUE;

			RASTERFOLIE:
				(* Virtuelle Masterachse *)
				axis_virt_master.st_config.b_config_fertig := FALSE;
				axis_virt_master.st_config.b_limitsensor_negativ_vorhanden := FALSE;
				axis_virt_master.st_config.b_limitsensor_positiv_vorhanden := FALSE;
				axis_virt_master.st_config.b_refsensor_vorhanden := FALSE;
				axis_virt_master.st_config.r_getriebefaktor := 1.0;
				axis_virt_master.st_config.i16_achstyp := RUND_VIRTUELL;
				axis_virt_master.st_config.i16_meld_startindex := 1400;
				axis_virt_master.st_config.s_beschreibung := ' ';
				axis_virt_master.st_config.s_instanz_name := 'Virtuelle Masterachse';
				axis_virt_master.st_config.ui16_ethercat_slave_id := 0;
				axis_virt_master.st_config.ui16_ethercat_adr := 0;
				axis_virt_master.st_config.b_config_fertig := TRUE;
				(* Bestueckachse *)
				axis_bestueckachse.st_config.b_config_fertig := FALSE;
				axis_bestueckachse.st_config.b_limitsensor_negativ_vorhanden := FALSE;
				axis_bestueckachse.st_config.b_limitsensor_positiv_vorhanden := FALSE;
				axis_bestueckachse.st_config.b_refsensor_vorhanden := FALSE;
				axis_bestueckachse.st_config.r_getriebefaktor := 1.0;
				axis_bestueckachse.st_config.i16_achstyp := RUND;
				axis_bestueckachse.st_config.i16_meld_startindex := 1000;
				axis_bestueckachse.st_config.s_beschreibung := ' ';
				axis_bestueckachse.st_config.s_instanz_name := 'Bestückachse';
				axis_bestueckachse.st_config.ui16_ethercat_slave_id := 2;
				axis_bestueckachse.st_config.ui16_ethercat_adr := 1010;
				axis_bestueckachse.st_config.b_config_fertig := TRUE;
				(* Z-Achse *)
				axis_z_achse.st_config.b_config_fertig := FALSE;
				axis_z_achse.st_config.b_limitsensor_negativ_vorhanden := TRUE;
				axis_z_achse.st_config.b_limitsensor_positiv_vorhanden := TRUE;
				axis_z_achse.st_config.b_refsensor_vorhanden := FALSE;
				axis_z_achse.st_config.r_getriebefaktor := 1.0;
				axis_z_achse.st_config.i16_achstyp := LINEAR;
				axis_z_achse.st_config.i16_meld_startindex := 1100;
				axis_z_achse.st_config.s_beschreibung := ' ';
				axis_z_achse.st_config.s_instanz_name := 'Z-Achse';
				axis_z_achse.st_config.ui16_ethercat_slave_id := 2;
				axis_z_achse.st_config.ui16_ethercat_adr := 1012;
				axis_z_achse.st_config.b_config_fertig := TRUE;
				(* Y-Achse *)
				axis_y_achse.st_config.b_config_fertig := FALSE;
				axis_y_achse.st_config.b_limitsensor_negativ_vorhanden := TRUE;
				axis_y_achse.st_config.b_limitsensor_positiv_vorhanden := TRUE;
				axis_y_achse.st_config.b_refsensor_vorhanden := FALSE;
				axis_y_achse.st_config.r_getriebefaktor := 1.0;
				axis_y_achse.st_config.i16_achstyp := LINEAR;
				axis_y_achse.st_config.i16_meld_startindex := 1200;
				axis_y_achse.st_config.s_beschreibung := ' ';
				axis_y_achse.st_config.s_instanz_name := 'Y-Achse';
				axis_y_achse.st_config.ui16_ethercat_slave_id := 2;
				axis_y_achse.st_config.ui16_ethercat_adr := 1012;
				axis_y_achse.st_config.b_config_fertig := TRUE;

		END_CASE
ELSE
	b_config_fertig := TRUE;
END_IF
END_PROGRAM

(* POU Gemeinsamkeiten17xx/Initialisierung/Startup/ST_Datainit_Fast_Zylinder, ST *)
PROGRAM ST_Datainit_Fast_Zylinder
VAR
	b_config_fertig			: BOOL := FALSE;
END_VAR
CASE gst_datensatz.st_md.i16_typ_zelle OF
	KEINE_ZELLE:
 		;
	BESTUECKZELLE_1700:
		IF 	NOT zyl_bandfaenger.fb.st_config.b_config_fertig OR
			NOT zyl_bandklemmen.fb.st_config.b_config_fertig OR
			NOT zyl_oelen_unten.fb.st_config.b_config_fertig OR
			NOT zyl_oelen_oben.fb.st_config.b_config_fertig THEN


					(*Banölen unten*)
					zyl_oelen_unten.fb.st_config.b_config_fertig := FALSE;
					zyl_oelen_unten.fb.st_config.b_endlage1_aktiv := FALSE;
					zyl_oelen_unten.fb.st_config.b_endlage2_aktiv := FALSE;
					zyl_oelen_unten.fb.st_config.b_sensor1_aktiv := FALSE;
					zyl_oelen_unten.fb.st_config.b_sensor2_aktiv := FALSE;
					zyl_oelen_unten.fb.st_config.i16_gruppe := 1;
					zyl_oelen_unten.fb.st_config.i16_identnummer :=45;
					zyl_oelen_unten.fb.st_config.i16_meld_startindex := 2880;
					zyl_oelen_unten.fb.st_config.str_beschreibung := ' ';
					zyl_oelen_unten.fb.st_config.str_instanz_name := 'Bandoelen unten';
					zyl_oelen_unten.fb.st_config.str_zylinder_typ := '1V2E_EIN_AUS'; (*1V2E_EIN_AUS*)
					zyl_oelen_unten.fb.st_config.t_ein_aus_fahrzeit := t#100ms;
					zyl_oelen_unten.fb.st_config.t_ueberwachungszeit := t#1500ms;
					zyl_oelen_unten.fb.st_config.i16_tzk_faktor_ausfahren := 100;
					zyl_oelen_unten.fb.st_config.i16_tzk_faktor_einfahren := 100;
					zyl_oelen_unten.fb.st_config.b_config_fertig := TRUE;

					(*Banölen oben*)
					zyl_oelen_oben.fb.st_config.b_config_fertig := FALSE;
					zyl_oelen_oben.fb.st_config.b_endlage1_aktiv := FALSE;
					zyl_oelen_oben.fb.st_config.b_endlage2_aktiv := FALSE;
					zyl_oelen_oben.fb.st_config.b_sensor1_aktiv := FALSE;
					zyl_oelen_oben.fb.st_config.b_sensor2_aktiv := FALSE;
					zyl_oelen_oben.fb.st_config.i16_gruppe := 1;
					zyl_oelen_oben.fb.st_config.i16_identnummer :=46 ;
					zyl_oelen_oben.fb.st_config.i16_meld_startindex := 2900;
					zyl_oelen_oben.fb.st_config.str_beschreibung := ' ';
					zyl_oelen_oben.fb.st_config.str_instanz_name := 'Bandoelen oben';
					zyl_oelen_oben.fb.st_config.str_zylinder_typ := '1V2E_EIN_AUS'; (*1V2E_EIN_AUS*)
					zyl_oelen_oben.fb.st_config.t_ein_aus_fahrzeit := t#100ms;
					zyl_oelen_oben.fb.st_config.t_ueberwachungszeit := t#1500ms;
					zyl_oelen_oben.fb.st_config.i16_tzk_faktor_ausfahren := 100;
					zyl_oelen_oben.fb.st_config.i16_tzk_faktor_einfahren := 100;
					zyl_oelen_oben.fb.st_config.b_config_fertig := TRUE;

				(* Abhängig vom Bandwechseltyp *)
				CASE gst_datensatz.st_wkz.i16_typ_bandeinzug OF
					KEIN_EINZUG:
						;

					STANDARD_2FACH_V2:
						;

					BANDWECHSLER_V2:
						(* 1700: Bandfaenger *)
						zyl_bandfaenger.fb.st_config.b_config_fertig := FALSE;
						zyl_bandfaenger.fb.st_config.b_endlage1_aktiv := FALSE;
						zyl_bandfaenger.fb.st_config.b_endlage2_aktiv := FALSE;
						zyl_bandfaenger.fb.st_config.b_sensor1_aktiv := FALSE;
						zyl_bandfaenger.fb.st_config.b_sensor2_aktiv := FALSE;
						zyl_bandfaenger.fb.st_config.i16_gruppe := 1;
						zyl_bandfaenger.fb.st_config.i16_identnummer := 5;
						zyl_bandfaenger.fb.st_config.i16_meld_startindex := 2080;
						zyl_bandfaenger.fb.st_config.str_beschreibung := ' ';
						zyl_bandfaenger.fb.st_config.str_instanz_name := 'Bandfänger';
						zyl_bandfaenger.fb.st_config.str_zylinder_typ := '1V0E_NO';
						zyl_bandfaenger.fb.st_config.t_ein_aus_fahrzeit := t#0ms;
						zyl_bandfaenger.fb.st_config.t_ueberwachungszeit := t#500ms;
						zyl_bandfaenger.fb.st_config.i16_tzk_faktor_ausfahren := 100;
						zyl_bandfaenger.fb.st_config.i16_tzk_faktor_einfahren := 100;
						zyl_bandfaenger.fb.st_config.b_config_fertig := TRUE;
						(* 1700: Bandklemmen *)
						zyl_bandklemmen.fb.st_config.b_config_fertig := FALSE;
						zyl_bandklemmen.fb.st_config.b_endlage1_aktiv := FALSE;
						zyl_bandklemmen.fb.st_config.b_endlage2_aktiv := FALSE;
						zyl_bandklemmen.fb.st_config.b_sensor1_aktiv := FALSE;
						zyl_bandklemmen.fb.st_config.b_sensor2_aktiv := FALSE;
						zyl_bandklemmen.fb.st_config.i16_gruppe := 1;
						zyl_bandklemmen.fb.st_config.i16_identnummer := 6;
						zyl_bandklemmen.fb.st_config.i16_meld_startindex := 2100;
						zyl_bandklemmen.fb.st_config.str_beschreibung := ' ';
						zyl_bandklemmen.fb.st_config.str_instanz_name := 'Bandklemmen';
						zyl_bandklemmen.fb.st_config.str_zylinder_typ := '1V0E_NO';
						zyl_bandklemmen.fb.st_config.t_ein_aus_fahrzeit := t#0ms;
						zyl_bandklemmen.fb.st_config.t_ueberwachungszeit := t#500ms;
						zyl_bandklemmen.fb.st_config.i16_tzk_faktor_ausfahren := 100;
						zyl_bandklemmen.fb.st_config.i16_tzk_faktor_einfahren := 100;
						zyl_bandklemmen.fb.st_config.b_config_fertig := TRUE;

					SERVO:
						;
				END_CASE
		ELSE
			b_config_fertig := FALSE;
		END_IF

	BESTUECKZELLE_1720:
		IF 	NOT zyl_bandfaenger_li.fb.st_config.b_config_fertig OR
			NOT zyl_bandfaenger_re.fb.st_config.b_config_fertig OR
			NOT zyl_bandklemmen_li.fb.st_config.b_config_fertig OR
			NOT zyl_bandklemmen_re.fb.st_config.b_config_fertig
			THEN
				(* Abhängig vom Bandwechseltyp *)
				CASE gst_datensatz.st_wkz.i16_typ_bandeinzug OF
					KEIN_EINZUG:
						;

					STANDARD_2FACH_V2:
						(* 1720: Bandfaenger links *)
						zyl_bandfaenger_li.fb.st_config.b_config_fertig := FALSE;
						zyl_bandfaenger_li.fb.st_config.b_endlage1_aktiv := FALSE;
						zyl_bandfaenger_li.fb.st_config.b_endlage2_aktiv := FALSE;
						zyl_bandfaenger_li.fb.st_config.b_sensor1_aktiv := FALSE;
						zyl_bandfaenger_li.fb.st_config.b_sensor2_aktiv := FALSE;
						zyl_bandfaenger_li.fb.st_config.i16_gruppe := 1;
						zyl_bandfaenger_li.fb.st_config.i16_identnummer := 1;
						zyl_bandfaenger_li.fb.st_config.i16_meld_startindex := 2000;
						zyl_bandfaenger_li.fb.st_config.str_beschreibung := ' ';
						zyl_bandfaenger_li.fb.st_config.str_instanz_name := 'Bandfänger links';
						zyl_bandfaenger_li.fb.st_config.str_zylinder_typ := '1V0E_NO';
						zyl_bandfaenger_li.fb.st_config.t_ein_aus_fahrzeit := t#0ms;
						zyl_bandfaenger_li.fb.st_config.t_ueberwachungszeit := t#500ms;
						zyl_bandfaenger_li.fb.st_config.i16_tzk_faktor_ausfahren := 100;
						zyl_bandfaenger_li.fb.st_config.i16_tzk_faktor_einfahren := 100;
						zyl_bandfaenger_li.fb.st_config.b_config_fertig := TRUE;
						(* 1720: Bandfaenger rechts *)
						zyl_bandfaenger_re.fb.st_config.b_config_fertig := FALSE;
						zyl_bandfaenger_re.fb.st_config.b_endlage1_aktiv := FALSE;
						zyl_bandfaenger_re.fb.st_config.b_endlage2_aktiv := FALSE;
						zyl_bandfaenger_re.fb.st_config.b_sensor1_aktiv := FALSE;
						zyl_bandfaenger_re.fb.st_config.b_sensor2_aktiv := FALSE;
						zyl_bandfaenger_re.fb.st_config.i16_gruppe := 1;
						zyl_bandfaenger_re.fb.st_config.i16_identnummer := 2;
						zyl_bandfaenger_re.fb.st_config.i16_meld_startindex := 2020;
						zyl_bandfaenger_re.fb.st_config.str_beschreibung := ' ';
						zyl_bandfaenger_re.fb.st_config.str_instanz_name := 'Bandfänger rechts';
						zyl_bandfaenger_re.fb.st_config.str_zylinder_typ := '1V0E_NO';
						zyl_bandfaenger_re.fb.st_config.t_ein_aus_fahrzeit := t#0ms;
						zyl_bandfaenger_re.fb.st_config.t_ueberwachungszeit := t#500ms;
						zyl_bandfaenger_re.fb.st_config.i16_tzk_faktor_ausfahren := 100;
						zyl_bandfaenger_re.fb.st_config.i16_tzk_faktor_einfahren := 100;
						zyl_bandfaenger_re.fb.st_config.b_config_fertig := TRUE;
						
						(* 1720: Bandklemmen links *)
						zyl_bandklemmen_li.fb.st_config.b_config_fertig := FALSE;
						zyl_bandklemmen_li.fb.st_config.b_endlage1_aktiv := FALSE;
						zyl_bandklemmen_li.fb.st_config.b_endlage2_aktiv := FALSE;
						zyl_bandklemmen_li.fb.st_config.b_sensor1_aktiv := FALSE;
						zyl_bandklemmen_li.fb.st_config.b_sensor2_aktiv := FALSE;
						zyl_bandklemmen_li.fb.st_config.i16_gruppe := 1;
						zyl_bandklemmen_li.fb.st_config.i16_identnummer := 3;
						zyl_bandklemmen_li.fb.st_config.i16_meld_startindex := 2040;
						zyl_bandklemmen_li.fb.st_config.str_beschreibung := ' ';
						zyl_bandklemmen_li.fb.st_config.str_instanz_name := 'Bandklemmen links';
						zyl_bandklemmen_li.fb.st_config.str_zylinder_typ := '1V0E_NO';
						zyl_bandklemmen_li.fb.st_config.t_ein_aus_fahrzeit := t#0ms;
						zyl_bandklemmen_li.fb.st_config.t_ueberwachungszeit := t#500ms;
						zyl_bandklemmen_li.fb.st_config.i16_tzk_faktor_ausfahren := 100;
						zyl_bandklemmen_li.fb.st_config.i16_tzk_faktor_einfahren := 100;
						zyl_bandklemmen_li.fb.st_config.b_config_fertig := TRUE;
						(* 1720: Bandklemmen rechts *)
						zyl_bandklemmen_re.fb.st_config.b_config_fertig := FALSE;
						zyl_bandklemmen_re.fb.st_config.b_endlage1_aktiv := FALSE;
						zyl_bandklemmen_re.fb.st_config.b_endlage2_aktiv := FALSE;
						zyl_bandklemmen_re.fb.st_config.b_sensor1_aktiv := FALSE;
						zyl_bandklemmen_re.fb.st_config.b_sensor2_aktiv := FALSE;
						zyl_bandklemmen_re.fb.st_config.i16_gruppe := 1;
						zyl_bandklemmen_re.fb.st_config.i16_identnummer := 4;
						zyl_bandklemmen_re.fb.st_config.i16_meld_startindex := 2060;
						zyl_bandklemmen_re.fb.st_config.str_beschreibung := ' ';
						zyl_bandklemmen_re.fb.st_config.str_instanz_name := 'Bandklemmen rechts';
						zyl_bandklemmen_re.fb.st_config.str_zylinder_typ := '1V0E_NO';
						zyl_bandklemmen_re.fb.st_config.t_ein_aus_fahrzeit := t#0ms;
						zyl_bandklemmen_re.fb.st_config.t_ueberwachungszeit := t#500ms;
						zyl_bandklemmen_re.fb.st_config.i16_tzk_faktor_ausfahren := 100;
						zyl_bandklemmen_re.fb.st_config.i16_tzk_faktor_einfahren := 100;
						zyl_bandklemmen_re.fb.st_config.b_config_fertig := TRUE;
				
					BANDWECHSLER_V2:
						;

					SERVO:
						;
				END_CASE;
		ELSE
			b_config_fertig := FALSE;
		END_IF

	RASTERFOLIE:
		;
END_CASE
END_PROGRAM

(* POU Gemeinsamkeiten17xx/Initialisierung/Startup/ST_Datainit_Stationen, ST *)
PROGRAM ST_Datainit_Stationen
VAR
	b_config_fertig			: BOOL := FALSE;
	i						: INT := 0;
	Index					: INT := 0;
END_VAR
IF	NOT betriebsarten.st_config.b_config_fertig OR
	NOT betriebsfreigaben.st_config.b_config_fertig OR
	NOT stoerungen_quittieren.st_config.b_config_fertig OR
	NOT bandeinzug_kontroller.st_config.b_config_fertig OR
	NOT wt_transport_kontroller.st_config.b_config_fertig OR
	NOT wt_transport_beladen.st_config.b_config_fertig OR
	NOT wt_transport_abgabe.st_config.b_config_fertig OR
	NOT routing_backpanel.st_config.b_config_fertig OR
	NOT routing_nachbarpc.st_config.b_config_fertig OR
	NOT UPS.st_config.b_config_fertig OR
	NOT haspel_kontroller.st_config.b_config_fertig OR
	NOT haspel_li.fb.st_config.b_config_fertig OR
	NOT haspel_re.fb.st_config.b_config_fertig OR
	NOT hublift_links.st_config.b_config_fertig OR
	NOT hublift_rechts.st_config.b_config_fertig OR
	NOT wkz_absicherung.st_config.b_config_fertig OR
	NOT stueckzahlen.fb.st_config.b_config_fertig OR
	NOT bandwechsel_kontroller.st_config.b_config_fertig OR
	NOT bandspruehoeler.st_config.b_config_fertig OR
	NOT einpresskraft_kontroller.st_config.b_config_fertig OR
	NOT kraftmessdose.fb.st_config.b_config_fertig OR
	NOT nockenschaltwerk_bestueckachse.st_config.b_config_fertig OR
	NOT safety.st_config.b_config_fertig OR
	NOT xml_server.st_config.b_config_fertig OR
	NOT fb_edit_mfps_bestuecken_z.st_config.b_config_fertig OR
	NOT fb_edit_mfps_bestuecken_y.st_config.b_config_fertig OR
	NOT fb_edit_mfps_yz_tisch.st_config.b_config_fertig OR
	NOT fb_camtable_bestueckachse.st_config.b_config_fertig OR
	NOT fb_edit_mfps_bestuecken_b.st_config.b_config_fertig OR
	NOT bbgen.st_config.b_config_fertig OR
	NOT barcode.fb.st_config.b_config_fertig OR
	NOT balluff_tag_reader.fb.st_config.b_config_fertig OR
	NOT wt_transport_warteposition_1720.st_config.b_config_fertig OR
	NOT wt_transport_beladen_1720.st_config.b_config_fertig OR
	NOT rasterfolienmontage.st_config.b_config_fertig OR
	NOT rasterfolieneinzug.st_config.b_config_fertig OR
	NOT Lesen_Schreiben_Tag.st_config.b_config_fertig OR
	NOT Service.st_config.b_config_fertig OR
	NOT ST_TouchProbe.st_config.b_config_fertig OR
	NOT wt_transport_warteposition_1700.st_config.b_config_fertig OR
	NOT wt_transport_beladen_achse_1700.st_config.b_config_fertig OR
	NOT EtherCatDiag[1].st_config.b_config_fertig
	THEN
		(* Betriebsarten *)
		betriebsarten.st_config.b_config_fertig := FALSE;
		betriebsarten.st_config.b_station_aktiv := TRUE;
		betriebsarten.st_config.i16_meld_startindex := 20;
		betriebsarten.st_config.str_beschreibung := ' ';
		betriebsarten.st_config.str_instanz_name := 'Betriebsarten';
		betriebsarten.st_config.b_config_fertig := TRUE;
		
		(* Betriebsfreigaben *)
		betriebsfreigaben.st_config.b_config_fertig := FALSE;
		betriebsfreigaben.st_config.b_station_aktiv := TRUE;
		betriebsfreigaben.st_config.i16_meld_startindex := 40;
		betriebsfreigaben.st_config.str_beschreibung := ' ';
		betriebsfreigaben.st_config.str_instanz_name := 'Betriebsfeigaben';
		betriebsfreigaben.st_config.b_config_fertig := TRUE;
		
		(* Störungen quittieren *)
		stoerungen_quittieren.st_config.b_config_fertig := FALSE;
		stoerungen_quittieren.st_config.b_station_aktiv := TRUE;
		stoerungen_quittieren.st_config.i16_meld_startindex := 60;
		stoerungen_quittieren.st_config.str_beschreibung := ' ';
		stoerungen_quittieren.st_config.str_instanz_name := 'Störungen quittieren';
		stoerungen_quittieren.st_config.b_config_fertig := TRUE;

		(* Bandeinzugskontroller *)
		bandeinzug_kontroller.st_config.b_config_fertig := FALSE;
		bandeinzug_kontroller.st_config.b_station_aktiv := TRUE;
		bandeinzug_kontroller.st_config.i16_meld_startindex := 80;
		bandeinzug_kontroller.st_config.str_beschreibung := ' ';
		bandeinzug_kontroller.st_config.str_instanz_name := 'Bandeinzugkontroller';
		bandeinzug_kontroller.st_config.b_config_fertig := TRUE;
		
		(* WT-Transport Kontroller *)
		wt_transport_kontroller.st_config.b_config_fertig := FALSE;
		wt_transport_kontroller.st_config.i16_meld_startindex := 100;
		wt_transport_kontroller.st_config.str_beschreibung := ' ';
		wt_transport_kontroller.st_config.str_instanz_name := 'WT-Transport Kontroller';
		wt_transport_kontroller.st_config.b_config_fertig := TRUE;
		
		(* WT-Transport Beladestation*)
		wt_transport_beladen.st_config.b_config_fertig := FALSE;
		wt_transport_beladen.st_config.i16_meld_startindex := 120;
		wt_transport_beladen.st_config.str_beschreibung := ' ';
		wt_transport_beladen.st_config.str_instanz_name := 'WT-Transport Beladestation';
		wt_transport_beladen.st_config.b_config_fertig := TRUE;
		
		(* WT-Transport Abgabestation *)
		wt_transport_abgabe.st_config.b_config_fertig := FALSE;
		wt_transport_abgabe.st_config.i16_meld_startindex := 140;
		wt_transport_abgabe.st_config.str_beschreibung := ' ';
		wt_transport_abgabe.st_config.str_instanz_name := 'WT-Transport Abgabestation';
		wt_transport_abgabe.st_config.b_config_fertig := TRUE;
		
		(* Routing Backpanel *)
		routing_backpanel.st_config.b_config_fertig := FALSE;
		routing_backpanel.st_config.i16_meld_startindex := 160;
		routing_backpanel.st_config.str_beschreibung := ' ';
		routing_backpanel.st_config.str_instanz_name := 'Routing Backpanel';
		routing_backpanel.st_config.b_config_fertig := TRUE;
		
		(* Routing Nachbar-PCs *)
		routing_nachbarpc.st_config.b_config_fertig := FALSE;
		routing_nachbarpc.st_config.i16_meld_startindex := 180;
		routing_nachbarpc.st_config.str_beschreibung := ' ';
		routing_nachbarpc.st_config.str_instanz_name := 'Routing Nachbar-PCs';
		routing_nachbarpc.st_config.b_config_fertig := TRUE;
		
		(* Haspelkontroller *)
		haspel_kontroller.st_config.b_config_fertig := FALSE;
		haspel_kontroller.st_config.b_station_aktiv := TRUE;
		haspel_kontroller.st_config.i16_meld_startindex := 200;
		haspel_kontroller.st_config.str_beschreibung := ' ';
		haspel_kontroller.st_config.str_instanz_name := 'Haspelkontroller';
		haspel_kontroller.t_abschaltzeit_motor := t#60s;
		haspel_kontroller.b_drehrichtung_antrieb_links := FALSE;
		haspel_kontroller.st_config.b_config_fertig := TRUE;

		(* Haspel links *)
		haspel_li.fb.st_config.b_config_fertig := FALSE;
		haspel_li.fb.st_config.b_station_aktiv := TRUE;
		haspel_li.fb.st_config.i16_meld_startindex := 220;
		haspel_li.fb.st_config.str_beschreibung := ' ';
		haspel_li.fb.st_config.str_instanz_name := 'Haspel links';
		haspel_li.fb.t_wartezeit_bandende := t#2s;
		haspel_li.fb.st_config.b_config_fertig := TRUE;
		
		(* Haspel rechts *)
		haspel_re.fb.st_config.b_config_fertig := FALSE;
		haspel_re.fb.st_config.b_station_aktiv := TRUE;
		haspel_re.fb.st_config.i16_meld_startindex := 240;
		haspel_re.fb.st_config.str_beschreibung := ' ';
		haspel_re.fb.st_config.str_instanz_name := 'Haspel rechts';
		haspel_re.fb.t_wartezeit_bandende := t#2s;
		haspel_re.fb.st_config.b_config_fertig := TRUE;
		
		(* Hublift links *)
		hublift_links.st_config.b_config_fertig := FALSE;
		hublift_links.st_config.i16_meld_startindex := 280;
		hublift_links.st_config.str_beschreibung := ' ';
		hublift_links.st_config.str_instanz_name := 'Hublift links';
		hublift_links.st_config.b_config_fertig := TRUE;
		
		(* Hublift rechts *)
		hublift_rechts.st_config.b_config_fertig := FALSE;
		hublift_rechts.st_config.i16_meld_startindex := 300;
		hublift_rechts.st_config.str_beschreibung := ' ';
		hublift_rechts.st_config.str_instanz_name := 'Hublift rechts';
		hublift_rechts.st_config.b_config_fertig := TRUE;
		
		(* Werkzeugabsicherung *)
		wkz_absicherung.st_config.b_config_fertig := FALSE;
		wkz_absicherung.st_config.b_station_aktiv := TRUE;
		wkz_absicherung.st_config.i16_meld_startindex := 320;
		wkz_absicherung.st_config.str_beschreibung := ' ';
		wkz_absicherung.st_config.str_instanz_name := 'Werkzeugabsicherung';
		wkz_absicherung.st_config.b_config_fertig := TRUE;
		
		(* Stückzahlen *)
		stueckzahlen.fb.st_config.b_config_fertig := FALSE;
		stueckzahlen.fb.st_config.b_station_aktiv := TRUE;
		stueckzahlen.fb.st_config.i16_meld_startindex := 340;
		stueckzahlen.fb.st_config.str_beschreibung := ' ';
		stueckzahlen.fb.st_config.str_instanz_name := 'Stueckzahlen';
		stueckzahlen.fb.st_config.b_config_fertig := TRUE;
		
		(* Bandwechselkontroller *)
		bandwechsel_kontroller.st_config.b_config_fertig := FALSE;
		bandwechsel_kontroller.st_config.b_station_aktiv := TRUE;
		bandwechsel_kontroller.st_config.i16_meld_startindex := 360;
		bandwechsel_kontroller.st_config.str_beschreibung := ' ';
		bandwechsel_kontroller.st_config.str_instanz_name := 'Bandwechselkontroller';
		bandwechsel_kontroller.st_config.b_config_fertig := TRUE;
		
		(* Bandsprühöler *)
		bandspruehoeler.st_config.b_config_fertig := FALSE;
		bandspruehoeler.st_config.b_station_aktiv := TRUE;
		bandspruehoeler.st_config.i16_meld_startindex := 380;
		bandspruehoeler.st_config.str_beschreibung := ' ';
		bandspruehoeler.st_config.str_instanz_name := 'Bandsprühöler';
		bandspruehoeler.st_config.b_config_fertig := TRUE;

